LIN {X 121.388,Y 125.417,Z 54.000,A 180.000,B 0.000,C 180.000} C_DIS
LIN {X 121.209,Y 125.491,Z 54.000,A 180.000,B 0.000,C 180.000} C_DIS
LIN {X 120.852,Y 125.619,Z 54.000,A 180.000,B 0.000,C 180.000} C_DIS
LIN {X 120.673,Y 125.674,Z 54.000,A 180.000,B 0.000,C 180.000} C_DIS
LIN {X 120.494,Y 125.726,Z 54.000,A 180.000,B 0.000,C 180.000} C_DIS
LIN {X 120.315,Y 125.774,Z 54.000,A 180.000,B 0.000,C 180.000} C_DIS
LIN {X 119.944,Y 125.857,Z 54.000,A 180.000,B 0.000,C 180.000} C_DIS
LIN {X 119.779,Y 125.886,Z 54.000,A 180.000,B 0.000,C 180.000} C_DIS
LIN {X 119.600,Y 125.914,Z 54.000,A 180.000,B 0.000,C 180.000} C_DIS
LIN {X 119.422,Y 125.941,Z 54.000,A 180.000,B 0.000,C 180.000} C_DIS
LIN {X 119.064,Y 125.975,Z 54.000,A 180.000,B 0.000,C 180.000} C_DIS
LIN {X 118.885,Y 125.987,Z 54.000,A 180.000,B 0.000,C 180.000} C_DIS
LIN {X 118.528,Y 125.998,Z 54.000,A 180.000,B 0.000,C 180.000} C_DIS
LIN {X 118.349,Y 125.994,Z 54.000,A 180.000,B 0.000,C 180.000} C_DIS
LIN {X 118.170,Y 125.988,Z 54.000,A 180.000,B 0.000,C 180.000} C_DIS
LIN {X 117.991,Y 125.980,Z 54.000,A 180.000,B 0.000,C 180.000} C_DIS
LIN {X 117.634,Y 125.947,Z 54.000,A 180.000,B 0.000,C 180.000} C_DIS
LIN {X 117.455,Y 125.923,Z 54.000,A 180.000,B 0.000,C 180.000} C_DIS
LIN {X 117.098,Y 125.866,Z 54.000,A 180.000,B 0.000,C 180.000} C_DIS
LIN {X 117.056,Y 125.857,Z 54.000,A 180.000,B 0.000,C 180.000} C_DIS
LIN {X 116.740,Y 125.787,Z 54.000,A 180.000,B 0.000,C 180.000} C_DIS
LIN {X 116.561,Y 125.742,Z 54.000,A 180.000,B 0.000,C 180.000} C_DIS
LIN {X 116.267,Y 125.656,Z 54.000,A 180.000,B 0.000,C 180.000} C_DIS
LIN {X 116.204,Y 125.638,Z 54.000,A 180.000,B 0.000,C 180.000} C_DIS
LIN {X 116.025,Y 125.575,Z 54.000,A 180.000,B 0.000,C 180.000} C_DIS
LIN {X 115.816,Y 125.500,Z 54.000,A 180.000,B 0.000,C 180.000} C_DIS
LIN {X 115.667,Y 125.441,Z 54.000,A 180.000,B 0.000,C 180.000} C_DIS
LIN {X 115.310,Y 125.286,Z 54.000,A 180.000,B 0.000,C 180.000} C_DIS
LIN {X 115.131,Y 125.195,Z 54.000,A 180.000,B 0.000,C 180.000} C_DIS
LIN {X 114.952,Y 125.104,Z 54.000,A 180.000,B 0.000,C 180.000} C_DIS
LIN {X 114.774,Y 125.004,Z 54.000,A 180.000,B 0.000,C 180.000} C_DIS
LIN {X 114.595,Y 124.898,Z 54.000,A 180.000,B 0.000,C 180.000} C_DIS
LIN {X 114.416,Y 124.787,Z 54.000,A 180.000,B 0.000,C 180.000} C_DIS
LIN {X 114.150,Y 124.606,Z 54.000,A 180.000,B 0.000,C 180.000} C_DIS
LIN {X 114.058,Y 124.540,Z 54.000,A 180.000,B 0.000,C 180.000} C_DIS
LIN {X 113.880,Y 124.402,Z 54.000,A 180.000,B 0.000,C 180.000} C_DIS
LIN {X 113.701,Y 124.261,Z 54.000,A 180.000,B 0.000,C 180.000} C_DIS
LIN {X 113.484,Y 124.070,Z 54.000,A 180.000,B 0.000,C 180.000} C_DIS
LIN {X 113.343,Y 123.943,Z 54.000,A 180.000,B 0.000,C 180.000} C_DIS
LIN {X 113.112,Y 123.712,Z 54.000,A 180.000,B 0.000,C 180.000} C_DIS
LIN {X 112.986,Y 123.579,Z 54.000,A 180.000,B 0.000,C 180.000} C_DIS
LIN {X 112.788,Y 123.354,Z 54.000,A 180.000,B 0.000,C 180.000} C_DIS
LIN {X 112.641,Y 123.176,Z 54.000,A 180.000,B 0.000,C 180.000} C_DIS
LIN {X 112.450,Y 122.928,Z 54.000,A 180.000,B 0.000,C 180.000} C_DIS
LIN {X 112.373,Y 122.818,Z 54.000,A 180.000,B 0.000,C 180.000} C_DIS
LIN {X 112.251,Y 122.639,Z 54.000,A 180.000,B 0.000,C 180.000} C_DIS
LIN {X 112.135,Y 122.461,Z 54.000,A 180.000,B 0.000,C 180.000} C_DIS
LIN {X 112.029,Y 122.282,Z 54.000,A 180.000,B 0.000,C 180.000} C_DIS
LIN {X 111.924,Y 122.103,Z 54.000,A 180.000,B 0.000,C 180.000} C_DIS
LIN {X 111.734,Y 121.731,Z 54.000,A 180.000,B 0.000,C 180.000} C_DIS
LIN {X 111.660,Y 121.567,Z 54.000,A 180.000,B 0.000,C 180.000} C_DIS
LIN {X 111.556,Y 121.325,Z 54.000,A 180.000,B 0.000,C 180.000} C_DIS
LIN {X 111.509,Y 121.209,Z 54.000,A 180.000,B 0.000,C 180.000} C_DIS
LIN {X 111.377,Y 120.841,Z 54.000,A 180.000,B 0.000,C 180.000} C_DIS
LIN {X 111.326,Y 120.673,Z 54.000,A 180.000,B 0.000,C 180.000} C_DIS
LIN {X 111.274,Y 120.494,Z 54.000,A 180.000,B 0.000,C 180.000} C_DIS
LIN {X 111.226,Y 120.315,Z 54.000,A 180.000,B 0.000,C 180.000} C_DIS
LIN {X 111.146,Y 119.958,Z 54.000,A 180.000,B 0.000,C 180.000} C_DIS
LIN {X 111.114,Y 119.779,Z 54.000,A 180.000,B 0.000,C 180.000} C_DIS
LIN {X 111.086,Y 119.600,Z 54.000,A 180.000,B 0.000,C 180.000} C_DIS
LIN {X 111.059,Y 119.422,Z 54.000,A 180.000,B 0.000,C 180.000} C_DIS
LIN {X 111.019,Y 119.006,Z 54.000,A 180.000,B 0.000,C 180.000} C_DIS
LIN {X 111.013,Y 118.885,Z 54.000,A 180.000,B 0.000,C 180.000} C_DIS
LIN {X 111.002,Y 118.528,Z 54.000,A 180.000,B 0.000,C 180.000} C_DIS
LIN {X 111.006,Y 118.349,Z 54.000,A 180.000,B 0.000,C 180.000} C_DIS
LIN {X 111.012,Y 118.170,Z 54.000,A 180.000,B 0.000,C 180.000} C_DIS
LIN {X 111.019,Y 117.994,Z 54.000,A 180.000,B 0.000,C 180.000} C_DIS
LIN {X 111.053,Y 117.634,Z 54.000,A 180.000,B 0.000,C 180.000} C_DIS
LIN {X 111.077,Y 117.455,Z 54.000,A 180.000,B 0.000,C 180.000} C_DIS
LIN {X 111.134,Y 117.098,Z 54.000,A 180.000,B 0.000,C 180.000} C_DIS
LIN {X 111.173,Y 116.919,Z 54.000,A 180.000,B 0.000,C 180.000} C_DIS
LIN {X 111.213,Y 116.740,Z 54.000,A 180.000,B 0.000,C 180.000} C_DIS
LIN {X 111.258,Y 116.561,Z 54.000,A 180.000,B 0.000,C 180.000} C_DIS
LIN {X 111.362,Y 116.204,Z 54.000,A 180.000,B 0.000,C 180.000} C_DIS
LIN {X 111.377,Y 116.159,Z 54.000,A 180.000,B 0.000,C 180.000} C_DIS
LIN {X 111.489,Y 115.846,Z 54.000,A 180.000,B 0.000,C 180.000} C_DIS
LIN {X 111.556,Y 115.675,Z 54.000,A 180.000,B 0.000,C 180.000} C_DIS
LIN {X 111.714,Y 115.310,Z 54.000,A 180.000,B 0.000,C 180.000} C_DIS
LIN {X 111.734,Y 115.269,Z 54.000,A 180.000,B 0.000,C 180.000} C_DIS
LIN {X 111.913,Y 114.918,Z 54.000,A 180.000,B 0.000,C 180.000} C_DIS
LIN {X 111.996,Y 114.774,Z 54.000,A 180.000,B 0.000,C 180.000} C_DIS
LIN {X 112.102,Y 114.595,Z 54.000,A 180.000,B 0.000,C 180.000} C_DIS
LIN {X 112.213,Y 114.416,Z 54.000,A 180.000,B 0.000,C 180.000} C_DIS
LIN {X 112.335,Y 114.237,Z 54.000,A 180.000,B 0.000,C 180.000} C_DIS
LIN {X 112.450,Y 114.072,Z 54.000,A 180.000,B 0.000,C 180.000} C_DIS
LIN {X 112.628,Y 113.841,Z 54.000,A 180.000,B 0.000,C 180.000} C_DIS
LIN {X 112.739,Y 113.701,Z 54.000,A 180.000,B 0.000,C 180.000} C_DIS
LIN {X 112.986,Y 113.421,Z 54.000,A 180.000,B 0.000,C 180.000} C_DIS
LIN {X 113.057,Y 113.343,Z 54.000,A 180.000,B 0.000,C 180.000} C_DIS
LIN {X 113.343,Y 113.057,Z 54.000,A 180.000,B 0.000,C 180.000} C_DIS
LIN {X 113.421,Y 112.986,Z 54.000,A 180.000,B 0.000,C 180.000} C_DIS
LIN {X 113.701,Y 112.739,Z 54.000,A 180.000,B 0.000,C 180.000} C_DIS
LIN {X 113.841,Y 112.628,Z 54.000,A 180.000,B 0.000,C 180.000} C_DIS
LIN {X 114.072,Y 112.450,Z 54.000,A 180.000,B 0.000,C 180.000} C_DIS
LIN {X 114.237,Y 112.335,Z 54.000,A 180.000,B 0.000,C 180.000} C_DIS
LIN {X 114.416,Y 112.213,Z 54.000,A 180.000,B 0.000,C 180.000} C_DIS
LIN {X 114.595,Y 112.102,Z 54.000,A 180.000,B 0.000,C 180.000} C_DIS
LIN {X 114.774,Y 111.996,Z 54.000,A 180.000,B 0.000,C 180.000} C_DIS
LIN {X 114.918,Y 111.913,Z 54.000,A 180.000,B 0.000,C 180.000} C_DIS
LIN {X 115.269,Y 111.734,Z 54.000,A 180.000,B 0.000,C 180.000} C_DIS
LIN {X 115.310,Y 111.714,Z 54.000,A 180.000,B 0.000,C 180.000} C_DIS
LIN {X 115.675,Y 111.556,Z 54.000,A 180.000,B 0.000,C 180.000} C_DIS
LIN {X 115.846,Y 111.489,Z 54.000,A 180.000,B 0.000,C 180.000} C_DIS
LIN {X 116.159,Y 111.377,Z 54.000,A 180.000,B 0.000,C 180.000} C_DIS
LIN {X 116.204,Y 111.362,Z 54.000,A 180.000,B 0.000,C 180.000} C_DIS
LIN {X 116.561,Y 111.258,Z 54.000,A 180.000,B 0.000,C 180.000} C_DIS
LIN {X 116.740,Y 111.213,Z 54.000,A 180.000,B 0.000,C 180.000} C_DIS
LIN {X 116.919,Y 111.173,Z 54.000,A 180.000,B 0.000,C 180.000} C_DIS
LIN {X 117.098,Y 111.134,Z 54.000,A 180.000,B 0.000,C 180.000} C_DIS
LIN {X 117.455,Y 111.077,Z 54.000,A 180.000,B 0.000,C 180.000} C_DIS
LIN {X 117.634,Y 111.053,Z 54.000,A 180.000,B 0.000,C 180.000} C_DIS
LIN {X 117.994,Y 111.019,Z 54.000,A 180.000,B 0.000,C 180.000} C_DIS
LIN {X 118.170,Y 111.012,Z 54.000,A 180.000,B 0.000,C 180.000} C_DIS
LIN {X 118.349,Y 111.006,Z 54.000,A 180.000,B 0.000,C 180.000} C_DIS
LIN {X 118.528,Y 111.002,Z 54.000,A 180.000,B 0.000,C 180.000} C_DIS
LIN {X 118.885,Y 111.013,Z 54.000,A 180.000,B 0.000,C 180.000} C_DIS
LIN {X 119.006,Y 111.019,Z 54.000,A 180.000,B 0.000,C 180.000} C_DIS
LIN {X 119.422,Y 111.059,Z 54.000,A 180.000,B 0.000,C 180.000} C_DIS
LIN {X 119.600,Y 111.086,Z 54.000,A 180.000,B 0.000,C 180.000} C_DIS
LIN {X 119.779,Y 111.114,Z 54.000,A 180.000,B 0.000,C 180.000} C_DIS
LIN {X 119.958,Y 111.146,Z 54.000,A 180.000,B 0.000,C 180.000} C_DIS
LIN {X 120.315,Y 111.226,Z 54.000,A 180.000,B 0.000,C 180.000} C_DIS
LIN {X 120.494,Y 111.274,Z 54.000,A 180.000,B 0.000,C 180.000} C_DIS
LIN {X 120.673,Y 111.326,Z 54.000,A 180.000,B 0.000,C 180.000} C_DIS
LIN {X 120.841,Y 111.377,Z 54.000,A 180.000,B 0.000,C 180.000} C_DIS
LIN {X 121.209,Y 111.509,Z 54.000,A 180.000,B 0.000,C 180.000} C_DIS
LIN {X 121.325,Y 111.556,Z 54.000,A 180.000,B 0.000,C 180.000} C_DIS
LIN {X 121.567,Y 111.660,Z 54.000,A 180.000,B 0.000,C 180.000} C_DIS
LIN {X 121.731,Y 111.734,Z 54.000,A 180.000,B 0.000,C 180.000} C_DIS
LIN {X 122.103,Y 111.924,Z 54.000,A 180.000,B 0.000,C 180.000} C_DIS
LIN {X 122.282,Y 112.029,Z 54.000,A 180.000,B 0.000,C 180.000} C_DIS
LIN {X 122.461,Y 112.135,Z 54.000,A 180.000,B 0.000,C 180.000} C_DIS
LIN {X 122.639,Y 112.251,Z 54.000,A 180.000,B 0.000,C 180.000} C_DIS
LIN {X 122.818,Y 112.373,Z 54.000,A 180.000,B 0.000,C 180.000} C_DIS
LIN {X 122.928,Y 112.450,Z 54.000,A 180.000,B 0.000,C 180.000} C_DIS
LIN {X 123.176,Y 112.641,Z 54.000,A 180.000,B 0.000,C 180.000} C_DIS
LIN {X 123.354,Y 112.788,Z 54.000,A 180.000,B 0.000,C 180.000} C_DIS
LIN {X 123.579,Y 112.986,Z 54.000,A 180.000,B 0.000,C 180.000} C_DIS
LIN {X 123.712,Y 113.112,Z 54.000,A 180.000,B 0.000,C 180.000} C_DIS
LIN {X 123.943,Y 113.343,Z 54.000,A 180.000,B 0.000,C 180.000} C_DIS
LIN {X 124.070,Y 113.484,Z 54.000,A 180.000,B 0.000,C 180.000} C_DIS
LIN {X 124.261,Y 113.701,Z 54.000,A 180.000,B 0.000,C 180.000} C_DIS
LIN {X 124.402,Y 113.880,Z 54.000,A 180.000,B 0.000,C 180.000} C_DIS
LIN {X 124.540,Y 114.058,Z 54.000,A 180.000,B 0.000,C 180.000} C_DIS
LIN {X 124.606,Y 114.150,Z 54.000,A 180.000,B 0.000,C 180.000} C_DIS
LIN {X 124.787,Y 114.416,Z 54.000,A 180.000,B 0.000,C 180.000} C_DIS
LIN {X 124.898,Y 114.595,Z 54.000,A 180.000,B 0.000,C 180.000} C_DIS
LIN {X 125.004,Y 114.774,Z 54.000,A 180.000,B 0.000,C 180.000} C_DIS
LIN {X 125.104,Y 114.952,Z 54.000,A 180.000,B 0.000,C 180.000} C_DIS
LIN {X 125.195,Y 115.131,Z 54.000,A 180.000,B 0.000,C 180.000} C_DIS
LIN {X 125.286,Y 115.310,Z 54.000,A 180.000,B 0.000,C 180.000} C_DIS
LIN {X 125.441,Y 115.667,Z 54.000,A 180.000,B 0.000,C 180.000} C_DIS
LIN {X 125.500,Y 115.816,Z 54.000,A 180.000,B 0.000,C 180.000} C_DIS
LIN {X 125.575,Y 116.025,Z 54.000,A 180.000,B 0.000,C 180.000} C_DIS
LIN {X 125.638,Y 116.204,Z 54.000,A 180.000,B 0.000,C 180.000} C_DIS
LIN {X 125.742,Y 116.561,Z 54.000,A 180.000,B 0.000,C 180.000} C_DIS
LIN {X 125.787,Y 116.740,Z 54.000,A 180.000,B 0.000,C 180.000} C_DIS
LIN {X 125.857,Y 117.056,Z 54.000,A 180.000,B 0.000,C 180.000} C_DIS
LIN {X 125.866,Y 117.098,Z 54.000,A 180.000,B 0.000,C 180.000} C_DIS
LIN {X 125.923,Y 117.455,Z 54.000,A 180.000,B 0.000,C 180.000} C_DIS
LIN {X 125.947,Y 117.634,Z 54.000,A 180.000,B 0.000,C 180.000} C_DIS
LIN {X 125.980,Y 117.991,Z 54.000,A 180.000,B 0.000,C 180.000} C_DIS
LIN {X 125.988,Y 118.170,Z 54.000,A 180.000,B 0.000,C 180.000} C_DIS
LIN {X 125.994,Y 118.349,Z 54.000,A 180.000,B 0.000,C 180.000} C_DIS
LIN {X 125.998,Y 118.528,Z 54.000,A 180.000,B 0.000,C 180.000} C_DIS
LIN {X 125.987,Y 118.885,Z 54.000,A 180.000,B 0.000,C 180.000} C_DIS
LIN {X 125.975,Y 119.064,Z 54.000,A 180.000,B 0.000,C 180.000} C_DIS
LIN {X 125.941,Y 119.422,Z 54.000,A 180.000,B 0.000,C 180.000} C_DIS
LIN {X 125.914,Y 119.600,Z 54.000,A 180.000,B 0.000,C 180.000} C_DIS
LIN {X 125.886,Y 119.779,Z 54.000,A 180.000,B 0.000,C 180.000} C_DIS
LIN {X 125.857,Y 119.944,Z 54.000,A 180.000,B 0.000,C 180.000} C_DIS
LIN {X 125.774,Y 120.315,Z 54.000,A 180.000,B 0.000,C 180.000} C_DIS
LIN {X 125.726,Y 120.494,Z 54.000,A 180.000,B 0.000,C 180.000} C_DIS
LIN {X 125.674,Y 120.673,Z 54.000,A 180.000,B 0.000,C 180.000} C_DIS
LIN {X 125.619,Y 120.852,Z 54.000,A 180.000,B 0.000,C 180.000} C_DIS
LIN {X 125.491,Y 121.209,Z 54.000,A 180.000,B 0.000,C 180.000} C_DIS
LIN {X 125.417,Y 121.388,Z 54.000,A 180.000,B 0.000,C 180.000} C_DIS
LIN {X 125.321,Y 121.610,Z 54.000,A 180.000,B 0.000,C 180.000} C_DIS
LIN {X 125.258,Y 121.746,Z 54.000,A 180.000,B 0.000,C 180.000} C_DIS
LIN {X 125.076,Y 122.103,Z 54.000,A 180.000,B 0.000,C 180.000} C_DIS
LIN {X 124.971,Y 122.282,Z 54.000,A 180.000,B 0.000,C 180.000} C_DIS
LIN {X 124.939,Y 122.336,Z 54.000,A 180.000,B 0.000,C 180.000} C_DIS
; Link Move Starts
LIN {X 124.773,Y 122.604,Z 54.000,A 180.000,B 0.000,C 180.000} C_DIS
LIN {X 124.596,Y 122.864,Z 53.999,A 180.000,B 0.000,C 180.000} C_DIS
LIN {X 124.406,Y 123.115,Z 53.998,A 180.000,B 0.000,C 180.000} C_DIS
LIN {X 124.207,Y 123.360,Z 53.996,A 180.000,B 0.000,C 180.000} C_DIS
LIN {X 123.999,Y 123.596,Z 53.994,A 180.000,B 0.000,C 180.000} C_DIS
LIN {X 123.778,Y 123.821,Z 53.991,A 180.000,B 0.000,C 180.000} C_DIS
LIN {X 123.551,Y 124.039,Z 53.988,A 180.000,B 0.000,C 180.000} C_DIS
LIN {X 123.315,Y 124.247,Z 53.985,A 180.000,B 0.000,C 180.000} C_DIS
LIN {X 123.068,Y 124.443,Z 53.981,A 180.000,B 0.000,C 180.000} C_DIS
LIN {X 122.814,Y 124.630,Z 53.977,A 180.000,B 0.000,C 180.000} C_DIS
LIN {X 122.554,Y 124.807,Z 53.972,A 180.000,B 0.000,C 180.000} C_DIS
LIN {X 122.420,Y 124.890,Z 53.969,A 180.000,B 0.000,C 180.000} C_DIS
LIN {X 122.284,Y 124.970,Z 53.967,A 180.000,B 0.000,C 180.000} C_DIS
LIN {X 122.149,Y 125.050,Z 53.964,A 180.000,B 0.000,C 180.000} C_DIS
LIN {X 122.009,Y 125.124,Z 53.961,A 180.000,B 0.000,C 180.000} C_DIS
LIN {X 121.869,Y 125.195,Z 53.959,A 180.000,B 0.000,C 180.000} C_DIS
LIN {X 121.729,Y 125.267,Z 53.956,A 180.000,B 0.000,C 180.000} C_DIS
LIN {X 121.585,Y 125.332,Z 53.952,A 180.000,B 0.000,C 180.000} C_DIS
LIN {X 121.441,Y 125.394,Z 53.949,A 180.000,B 0.000,C 180.000} C_DIS
LIN {X 121.296,Y 125.457,Z 53.946,A 180.000,B 0.000,C 180.000} C_DIS
LIN {X 121.149,Y 125.512,Z 53.943,A 180.000,B 0.000,C 180.000} C_DIS
LIN {X 121.001,Y 125.566,Z 53.939,A 180.000,B 0.000,C 180.000} C_DIS
LIN {X 120.852,Y 125.619,Z 53.936,A 180.000,B 0.000,C 180.000} C_DIS
LIN {X 120.702,Y 125.665,Z 53.932,A 180.000,B 0.000,C 180.000} C_DIS
LIN {X 120.551,Y 125.709,Z 53.928,A 180.000,B 0.000,C 180.000} C_DIS
LIN {X 120.399,Y 125.753,Z 53.925,A 180.000,B 0.000,C 180.000} C_DIS
LIN {X 120.246,Y 125.790,Z 53.921,A 180.000,B 0.000,C 180.000} C_DIS
LIN {X 120.092,Y 125.824,Z 53.917,A 180.000,B 0.000,C 180.000} C_DIS
LIN {X 119.939,Y 125.858,Z 53.913,A 180.000,B 0.000,C 180.000} C_DIS
LIN {X 119.784,Y 125.885,Z 53.909,A 180.000,B 0.000,C 180.000} C_DIS
LIN {X 119.628,Y 125.910,Z 53.905,A 180.000,B 0.000,C 180.000} C_DIS
LIN {X 119.472,Y 125.934,Z 53.900,A 180.000,B 0.000,C 180.000} C_DIS
LIN {X 119.316,Y 125.951,Z 53.896,A 180.000,B 0.000,C 180.000} C_DIS
LIN {X 119.159,Y 125.966,Z 53.892,A 180.000,B 0.000,C 180.000} C_DIS
LIN {X 119.002,Y 125.981,Z 53.887,A 180.000,B 0.000,C 180.000} C_DIS
LIN {X 118.845,Y 125.988,Z 53.883,A 180.000,B 0.000,C 180.000} C_DIS
LIN {X 118.687,Y 125.993,Z 53.878,A 180.000,B 0.000,C 180.000} C_DIS
LIN {X 118.530,Y 125.998,Z 53.873,A 180.000,B 0.000,C 180.000} C_DIS
LIN {X 118.373,Y 125.995,Z 53.869,A 180.000,B 0.000,C 180.000} C_DIS
LIN {X 118.215,Y 125.990,Z 53.864,A 180.000,B 0.000,C 180.000} C_DIS
LIN {X 118.058,Y 125.985,Z 53.859,A 180.000,B 0.000,C 180.000} C_DIS
LIN {X 117.901,Y 125.972,Z 53.854,A 180.000,B 0.000,C 180.000} C_DIS
LIN {X 117.822,Y 125.964,Z 53.851,A 180.000,B 0.000,C 180.000} C_DIS
LIN {X 117.744,Y 125.957,Z 53.849,A 180.000,B 0.000,C 180.000} C_DIS
LIN {X 117.666,Y 125.950,Z 53.846,A 180.000,B 0.000,C 180.000} C_DIS
LIN {X 117.587,Y 125.942,Z 53.844,A 180.000,B 0.000,C 180.000} C_DIS
LIN {X 117.509,Y 125.932,Z 53.841,A 180.000,B 0.000,C 180.000} C_DIS
LIN {X 117.431,Y 125.919,Z 53.839,A 180.000,B 0.000,C 180.000} C_DIS
LIN {X 117.354,Y 125.907,Z 53.836,A 180.000,B 0.000,C 180.000} C_DIS
LIN {X 117.198,Y 125.882,Z 53.831,A 180.000,B 0.000,C 180.000} C_DIS
LIN {X 117.120,Y 125.870,Z 53.828,A 180.000,B 0.000,C 180.000} C_DIS
LIN {X 117.043,Y 125.854,Z 53.825,A 180.000,B 0.000,C 180.000} C_DIS
LIN {X 116.889,Y 125.820,Z 53.820,A 180.000,B 0.000,C 180.000} C_DIS
LIN {X 116.736,Y 125.786,Z 53.815,A 180.000,B 0.000,C 180.000} C_DIS
LIN {X 116.659,Y 125.768,Z 53.812,A 180.000,B 0.000,C 180.000} C_DIS
LIN {X 116.583,Y 125.748,Z 53.809,A 180.000,B 0.000,C 180.000} C_DIS
LIN {X 116.507,Y 125.726,Z 53.806,A 180.000,B 0.000,C 180.000} C_DIS
LIN {X 116.356,Y 125.682,Z 53.801,A 180.000,B 0.000,C 180.000} C_DIS
LIN {X 116.205,Y 125.638,Z 53.796,A 180.000,B 0.000,C 180.000} C_DIS
LIN {X 116.130,Y 125.613,Z 53.793,A 180.000,B 0.000,C 180.000} C_DIS
LIN {X 115.982,Y 125.559,Z 53.787,A 180.000,B 0.000,C 180.000} C_DIS
LIN {X 115.908,Y 125.533,Z 53.785,A 180.000,B 0.000,C 180.000} C_DIS
LIN {X 115.759,Y 125.479,Z 53.779,A 180.000,B 0.000,C 180.000} C_DIS
LIN {X 115.687,Y 125.449,Z 53.776,A 180.000,B 0.000,C 180.000} C_DIS
LIN {X 115.614,Y 125.418,Z 53.774,A 180.000,B 0.000,C 180.000} C_DIS
LIN {X 115.470,Y 125.355,Z 53.768,A 180.000,B 0.000,C 180.000} C_DIS
LIN {X 115.325,Y 125.293,Z 53.763,A 180.000,B 0.000,C 180.000} C_DIS
LIN {X 115.255,Y 125.258,Z 53.760,A 180.000,B 0.000,C 180.000} C_DIS
LIN {X 115.114,Y 125.187,Z 53.754,A 180.000,B 0.000,C 180.000} C_DIS
LIN {X 115.044,Y 125.151,Z 53.752,A 180.000,B 0.000,C 180.000} C_DIS
LIN {X 114.904,Y 125.080,Z 53.746,A 180.000,B 0.000,C 180.000} C_DIS
LIN {X 114.835,Y 125.040,Z 53.743,A 180.000,B 0.000,C 180.000} C_DIS
LIN {X 114.768,Y 125.000,Z 53.741,A 180.000,B 0.000,C 180.000} C_DIS
LIN {X 114.632,Y 124.920,Z 53.735,A 180.000,B 0.000,C 180.000} C_DIS
LIN {X 114.496,Y 124.840,Z 53.730,A 180.000,B 0.000,C 180.000} C_DIS
LIN {X 114.431,Y 124.797,Z 53.727,A 180.000,B 0.000,C 180.000} C_DIS
LIN {X 114.300,Y 124.708,Z 53.721,A 180.000,B 0.000,C 180.000} C_DIS
LIN {X 114.235,Y 124.664,Z 53.719,A 180.000,B 0.000,C 180.000} C_DIS
LIN {X 114.105,Y 124.575,Z 53.713,A 180.000,B 0.000,C 180.000} C_DIS
LIN {X 114.042,Y 124.528,Z 53.710,A 180.000,B 0.000,C 180.000} C_DIS
LIN {X 113.980,Y 124.479,Z 53.708,A 180.000,B 0.000,C 180.000} C_DIS
LIN {X 113.855,Y 124.383,Z 53.702,A 180.000,B 0.000,C 180.000} C_DIS
LIN {X 113.731,Y 124.286,Z 53.697,A 180.000,B 0.000,C 180.000} C_DIS
LIN {X 113.671,Y 124.235,Z 53.694,A 180.000,B 0.000,C 180.000} C_DIS
LIN {X 113.553,Y 124.131,Z 53.688,A 180.000,B 0.000,C 180.000} C_DIS
LIN {X 113.494,Y 124.079,Z 53.686,A 180.000,B 0.000,C 180.000} C_DIS
LIN {X 113.376,Y 123.975,Z 53.680,A 180.000,B 0.000,C 180.000} C_DIS
LIN {X 113.320,Y 123.919,Z 53.677,A 180.000,B 0.000,C 180.000} C_DIS
LIN {X 113.208,Y 123.808,Z 53.672,A 180.000,B 0.000,C 180.000} C_DIS
LIN {X 113.097,Y 123.697,Z 53.666,A 180.000,B 0.000,C 180.000} C_DIS
LIN {X 113.041,Y 123.641,Z 53.664,A 180.000,B 0.000,C 180.000} C_DIS
LIN {X 112.989,Y 123.582,Z 53.661,A 180.000,B 0.000,C 180.000} C_DIS
LIN {X 112.728,Y 123.287,Z 53.647,A 180.000,B 0.000,C 180.000} C_DIS
LIN {X 112.680,Y 123.225,Z 53.644,A 180.000,B 0.000,C 180.000} C_DIS
LIN {X 112.583,Y 123.101,Z 53.639,A 180.000,B 0.000,C 180.000} C_DIS
LIN {X 112.438,Y 122.914,Z 53.631,A 180.000,B 0.000,C 180.000} C_DIS
LIN {X 112.394,Y 122.849,Z 53.628,A 180.000,B 0.000,C 180.000} C_DIS
LIN {X 112.172,Y 122.523,Z 53.614,A 180.000,B 0.000,C 180.000} C_DIS
LIN {X 112.132,Y 122.456,Z 53.611,A 180.000,B 0.000,C 180.000} C_DIS
LIN {X 112.011,Y 122.252,Z 53.603,A 180.000,B 0.000,C 180.000} C_DIS
LIN {X 111.931,Y 122.117,Z 53.598,A 180.000,B 0.000,C 180.000} C_DIS
LIN {X 111.895,Y 122.047,Z 53.595,A 180.000,B 0.000,C 180.000} C_DIS
LIN {X 111.716,Y 121.696,Z 53.581,A 180.000,B 0.000,C 180.000} C_DIS
LIN {X 111.685,Y 121.624,Z 53.578,A 180.000,B 0.000,C 180.000} C_DIS
LIN {X 111.529,Y 121.262,Z 53.565,A 180.000,B 0.000,C 180.000} C_DIS
LIN {X 111.502,Y 121.188,Z 53.562,A 180.000,B 0.000,C 180.000} C_DIS
LIN {X 111.368,Y 120.818,Z 53.548,A 180.000,B 0.000,C 180.000} C_DIS
LIN {X 111.346,Y 120.742,Z 53.545,A 180.000,B 0.000,C 180.000} C_DIS
LIN {X 111.259,Y 120.440,Z 53.534,A 180.000,B 0.000,C 180.000} C_DIS
LIN {X 111.237,Y 120.364,Z 53.532,A 180.000,B 0.000,C 180.000} C_DIS
LIN {X 111.151,Y 119.980,Z 53.518,A 180.000,B 0.000,C 180.000} C_DIS
LIN {X 111.134,Y 119.903,Z 53.515,A 180.000,B 0.000,C 180.000} C_DIS
LIN {X 111.072,Y 119.514,Z 53.501,A 180.000,B 0.000,C 180.000} C_DIS
LIN {X 111.060,Y 119.436,Z 53.499,A 180.000,B 0.000,C 180.000} C_DIS
LIN {X 111.023,Y 119.044,Z 53.485,A 180.000,B 0.000,C 180.000} C_DIS
LIN {X 111.016,Y 118.965,Z 53.482,A 180.000,B 0.000,C 180.000} C_DIS
LIN {X 111.003,Y 118.572,Z 53.468,A 180.000,B 0.000,C 180.000} C_DIS
LIN {X 111.001,Y 118.493,Z 53.466,A 180.000,B 0.000,C 180.000} C_DIS
LIN {X 111.014,Y 118.100,Z 53.452,A 180.000,B 0.000,C 180.000} C_DIS
LIN {X 111.017,Y 118.021,Z 53.449,A 180.000,B 0.000,C 180.000} C_DIS
LIN {X 111.054,Y 117.629,Z 53.435,A 180.000,B 0.000,C 180.000} C_DIS
LIN {X 111.062,Y 117.550,Z 53.433,A 180.000,B 0.000,C 180.000} C_DIS
LIN {X 111.123,Y 117.162,Z 53.419,A 180.000,B 0.000,C 180.000} C_DIS
LIN {X 111.137,Y 117.084,Z 53.416,A 180.000,B 0.000,C 180.000} C_DIS
LIN {X 111.222,Y 116.700,Z 53.402,A 180.000,B 0.000,C 180.000} C_DIS
LIN {X 111.240,Y 116.623,Z 53.400,A 180.000,B 0.000,C 180.000} C_DIS
LIN {X 111.306,Y 116.396,Z 53.391,A 180.000,B 0.000,C 180.000} C_DIS
LIN {X 111.350,Y 116.245,Z 53.386,A 180.000,B 0.000,C 180.000} C_DIS
LIN {X 111.373,Y 116.169,Z 53.383,A 180.000,B 0.000,C 180.000} C_DIS
LIN {X 111.506,Y 115.799,Z 53.369,A 180.000,B 0.000,C 180.000} C_DIS
LIN {X 111.534,Y 115.725,Z 53.367,A 180.000,B 0.000,C 180.000} C_DIS
LIN {X 111.628,Y 115.508,Z 53.358,A 180.000,B 0.000,C 180.000} C_DIS
LIN {X 111.690,Y 115.364,Z 53.353,A 180.000,B 0.000,C 180.000} C_DIS
LIN {X 111.723,Y 115.292,Z 53.350,A 180.000,B 0.000,C 180.000} C_DIS
LIN {X 111.901,Y 114.941,Z 53.336,A 180.000,B 0.000,C 180.000} C_DIS
LIN {X 111.938,Y 114.871,Z 53.334,A 180.000,B 0.000,C 180.000} C_DIS
LIN {X 112.018,Y 114.736,Z 53.328,A 180.000,B 0.000,C 180.000} C_DIS
LIN {X 112.139,Y 114.533,Z 53.320,A 180.000,B 0.000,C 180.000} C_DIS
LIN {X 112.180,Y 114.465,Z 53.317,A 180.000,B 0.000,C 180.000} C_DIS
LIN {X 112.401,Y 114.140,Z 53.303,A 180.000,B 0.000,C 180.000} C_DIS
LIN {X 112.447,Y 114.075,Z 53.301,A 180.000,B 0.000,C 180.000} C_DIS
LIN {X 112.543,Y 113.951,Z 53.295,A 180.000,B 0.000,C 180.000} C_DIS
LIN {X 112.688,Y 113.764,Z 53.287,A 180.000,B 0.000,C 180.000} C_DIS
LIN {X 112.737,Y 113.703,Z 53.284,A 180.000,B 0.000,C 180.000} C_DIS
LIN {X 112.894,Y 113.526,Z 53.276,A 180.000,B 0.000,C 180.000} C_DIS
LIN {X 112.998,Y 113.407,Z 53.270,A 180.000,B 0.000,C 180.000} C_DIS
LIN {X 113.051,Y 113.349,Z 53.268,A 180.000,B 0.000,C 180.000} C_DIS
LIN {X 113.162,Y 113.238,Z 53.262,A 180.000,B 0.000,C 180.000} C_DIS
LIN {X 113.329,Y 113.071,Z 53.254,A 180.000,B 0.000,C 180.000} C_DIS
LIN {X 113.386,Y 113.016,Z 53.251,A 180.000,B 0.000,C 180.000} C_DIS
LIN {X 113.563,Y 112.860,Z 53.243,A 180.000,B 0.000,C 180.000} C_DIS
LIN {X 113.682,Y 112.756,Z 53.237,A 180.000,B 0.000,C 180.000} C_DIS
LIN {X 113.742,Y 112.705,Z 53.235,A 180.000,B 0.000,C 180.000} C_DIS
LIN {X 113.866,Y 112.609,Z 53.229,A 180.000,B 0.000,C 180.000} C_DIS
LIN {X 114.053,Y 112.464,Z 53.221,A 180.000,B 0.000,C 180.000} C_DIS
LIN {X 114.116,Y 112.417,Z 53.218,A 180.000,B 0.000,C 180.000} C_DIS
LIN {X 114.312,Y 112.284,Z 53.210,A 180.000,B 0.000,C 180.000} C_DIS
LIN {X 114.442,Y 112.196,Z 53.204,A 180.000,B 0.000,C 180.000} C_DIS
LIN {X 114.508,Y 112.153,Z 53.202,A 180.000,B 0.000,C 180.000} C_DIS
LIN {X 114.644,Y 112.073,Z 53.196,A 180.000,B 0.000,C 180.000} C_DIS
LIN {X 114.779,Y 111.993,Z 53.191,A 180.000,B 0.000,C 180.000} C_DIS
LIN {X 114.847,Y 111.953,Z 53.188,A 180.000,B 0.000,C 180.000} C_DIS
LIN {X 114.916,Y 111.914,Z 53.185,A 180.000,B 0.000,C 180.000} C_DIS
LIN {X 115.056,Y 111.843,Z 53.180,A 180.000,B 0.000,C 180.000} C_DIS
LIN {X 115.196,Y 111.771,Z 53.174,A 180.000,B 0.000,C 180.000} C_DIS
LIN {X 115.267,Y 111.736,Z 53.172,A 180.000,B 0.000,C 180.000} C_DIS
LIN {X 115.338,Y 111.702,Z 53.169,A 180.000,B 0.000,C 180.000} C_DIS
LIN {X 115.482,Y 111.639,Z 53.164,A 180.000,B 0.000,C 180.000} C_DIS
LIN {X 115.555,Y 111.608,Z 53.161,A 180.000,B 0.000,C 180.000} C_DIS
LIN {X 115.627,Y 111.577,Z 53.159,A 180.000,B 0.000,C 180.000} C_DIS
LIN {X 115.699,Y 111.545,Z 53.156,A 180.000,B 0.000,C 180.000} C_DIS
LIN {X 115.772,Y 111.516,Z 53.154,A 180.000,B 0.000,C 180.000} C_DIS
LIN {X 115.846,Y 111.489,Z 53.151,A 180.000,B 0.000,C 180.000} C_DIS
LIN {X 115.920,Y 111.463,Z 53.149,A 180.000,B 0.000,C 180.000} C_DIS
LIN {X 116.069,Y 111.409,Z 53.144,A 180.000,B 0.000,C 180.000} C_DIS
LIN {X 116.217,Y 111.358,Z 53.139,A 180.000,B 0.000,C 180.000} C_DIS
LIN {X 116.369,Y 111.314,Z 53.134,A 180.000,B 0.000,C 180.000} C_DIS
LIN {X 116.520,Y 111.270,Z 53.129,A 180.000,B 0.000,C 180.000} C_DIS
LIN {X 116.672,Y 111.229,Z 53.124,A 180.000,B 0.000,C 180.000} C_DIS
LIN {X 116.826,Y 111.194,Z 53.120,A 180.000,B 0.000,C 180.000} C_DIS
LIN {X 116.979,Y 111.160,Z 53.115,A 180.000,B 0.000,C 180.000} C_DIS
LIN {X 117.133,Y 111.128,Z 53.111,A 180.000,B 0.000,C 180.000} C_DIS
LIN {X 117.289,Y 111.103,Z 53.106,A 180.000,B 0.000,C 180.000} C_DIS
LIN {X 117.445,Y 111.079,Z 53.102,A 180.000,B 0.000,C 180.000} C_DIS
LIN {X 117.601,Y 111.057,Z 53.097,A 180.000,B 0.000,C 180.000} C_DIS
LIN {X 117.757,Y 111.042,Z 53.093,A 180.000,B 0.000,C 180.000} C_DIS
LIN {X 117.914,Y 111.027,Z 53.089,A 180.000,B 0.000,C 180.000} C_DIS
LIN {X 118.071,Y 111.015,Z 53.085,A 180.000,B 0.000,C 180.000} C_DIS
LIN {X 118.229,Y 111.010,Z 53.081,A 180.000,B 0.000,C 180.000} C_DIS
LIN {X 118.386,Y 111.005,Z 53.077,A 180.000,B 0.000,C 180.000} C_DIS
LIN {X 118.544,Y 111.003,Z 53.073,A 180.000,B 0.000,C 180.000} C_DIS
LIN {X 118.701,Y 111.008,Z 53.070,A 180.000,B 0.000,C 180.000} C_DIS
LIN {X 118.858,Y 111.012,Z 53.066,A 180.000,B 0.000,C 180.000} C_DIS
LIN {X 119.016,Y 111.020,Z 53.062,A 180.000,B 0.000,C 180.000} C_DIS
LIN {X 119.172,Y 111.035,Z 53.059,A 180.000,B 0.000,C 180.000} C_DIS
LIN {X 119.329,Y 111.050,Z 53.056,A 180.000,B 0.000,C 180.000} C_DIS
LIN {X 119.486,Y 111.068,Z 53.052,A 180.000,B 0.000,C 180.000} C_DIS
LIN {X 119.641,Y 111.092,Z 53.049,A 180.000,B 0.000,C 180.000} C_DIS
LIN {X 119.797,Y 111.117,Z 53.046,A 180.000,B 0.000,C 180.000} C_DIS
LIN {X 119.952,Y 111.145,Z 53.043,A 180.000,B 0.000,C 180.000} C_DIS
LIN {X 120.106,Y 111.179,Z 53.040,A 180.000,B 0.000,C 180.000} C_DIS
LIN {X 120.259,Y 111.213,Z 53.037,A 180.000,B 0.000,C 180.000} C_DIS
LIN {X 120.412,Y 111.251,Z 53.034,A 180.000,B 0.000,C 180.000} C_DIS
LIN {X 120.564,Y 111.295,Z 53.032,A 180.000,B 0.000,C 180.000} C_DIS
LIN {X 120.715,Y 111.338,Z 53.029,A 180.000,B 0.000,C 180.000} C_DIS
LIN {X 120.865,Y 111.385,Z 53.027,A 180.000,B 0.000,C 180.000} C_DIS
LIN {X 121.161,Y 111.492,Z 53.022,A 180.000,B 0.000,C 180.000} C_DIS
LIN {X 121.453,Y 111.611,Z 53.018,A 180.000,B 0.000,C 180.000} C_DIS
LIN {X 121.741,Y 111.739,Z 53.014,A 180.000,B 0.000,C 180.000} C_DIS
LIN {X 122.021,Y 111.882,Z 53.011,A 180.000,B 0.000,C 180.000} C_DIS
LIN {X 122.296,Y 112.037,Z 53.008,A 180.000,B 0.000,C 180.000} C_DIS
LIN {X 122.565,Y 112.200,Z 53.005,A 180.000,B 0.000,C 180.000} C_DIS
LIN {X 122.826,Y 112.378,Z 53.003,A 180.000,B 0.000,C 180.000} C_DIS
LIN {X 123.078,Y 112.566,Z 53.002,A 180.000,B 0.000,C 180.000} C_DIS
LIN {X 123.325,Y 112.762,Z 53.001,A 180.000,B 0.000,C 180.000} C_DIS
LIN {X 123.561,Y 112.970,Z 53.000,A 180.000,B 0.000,C 180.000} C_DIS
LIN {X 123.729,Y 113.130,Z 53.000,A 180.000,B 0.000,C 180.000} C_DIS
; Cutting Move Starts
LIN {X 123.943,Y 113.343,Z 53.000,A 180.000,B 0.000,C 180.000} C_DIS
LIN {X 124.070,Y 113.484,Z 53.000,A 180.000,B 0.000,C 180.000} C_DIS
LIN {X 124.261,Y 113.701,Z 53.000,A 180.000,B 0.000,C 180.000} C_DIS
LIN {X 124.402,Y 113.880,Z 53.000,A 180.000,B 0.000,C 180.000} C_DIS
LIN {X 124.540,Y 114.058,Z 53.000,A 180.000,B 0.000,C 180.000} C_DIS
LIN {X 124.606,Y 114.150,Z 53.000,A 180.000,B 0.000,C 180.000} C_DIS
LIN {X 124.787,Y 114.416,Z 53.000,A 180.000,B 0.000,C 180.000} C_DIS
LIN {X 124.898,Y 114.595,Z 53.000,A 180.000,B 0.000,C 180.000} C_DIS
LIN {X 125.004,Y 114.774,Z 53.000,A 180.000,B 0.000,C 180.000} C_DIS
LIN {X 125.104,Y 114.952,Z 53.000,A 180.000,B 0.000,C 180.000} C_DIS
LIN {X 125.195,Y 115.131,Z 53.000,A 180.000,B 0.000,C 180.000} C_DIS
LIN {X 125.286,Y 115.310,Z 53.000,A 180.000,B 0.000,C 180.000} C_DIS
LIN {X 125.441,Y 115.667,Z 53.000,A 180.000,B 0.000,C 180.000} C_DIS
LIN {X 125.500,Y 115.816,Z 53.000,A 180.000,B 0.000,C 180.000} C_DIS
LIN {X 125.575,Y 116.025,Z 53.000,A 180.000,B 0.000,C 180.000} C_DIS
LIN {X 125.638,Y 116.204,Z 53.000,A 180.000,B 0.000,C 180.000} C_DIS
LIN {X 125.742,Y 116.561,Z 53.000,A 180.000,B 0.000,C 180.000} C_DIS
LIN {X 125.787,Y 116.740,Z 53.000,A 180.000,B 0.000,C 180.000} C_DIS
LIN {X 125.857,Y 117.056,Z 53.000,A 180.000,B 0.000,C 180.000} C_DIS
LIN {X 125.866,Y 117.098,Z 53.000,A 180.000,B 0.000,C 180.000} C_DIS
LIN {X 125.923,Y 117.455,Z 53.000,A 180.000,B 0.000,C 180.000} C_DIS
LIN {X 125.947,Y 117.634,Z 53.000,A 180.000,B 0.000,C 180.000} C_DIS
LIN {X 125.980,Y 117.991,Z 53.000,A 180.000,B 0.000,C 180.000} C_DIS
LIN {X 125.988,Y 118.170,Z 53.000,A 180.000,B 0.000,C 180.000} C_DIS
LIN {X 125.994,Y 118.349,Z 53.000,A 180.000,B 0.000,C 180.000} C_DIS
LIN {X 125.998,Y 118.528,Z 53.000,A 180.000,B 0.000,C 180.000} C_DIS
LIN {X 125.987,Y 118.885,Z 53.000,A 180.000,B 0.000,C 180.000} C_DIS
LIN {X 125.975,Y 119.064,Z 53.000,A 180.000,B 0.000,C 180.000} C_DIS
LIN {X 125.941,Y 119.422,Z 53.000,A 180.000,B 0.000,C 180.000} C_DIS
LIN {X 125.914,Y 119.600,Z 53.000,A 180.000,B 0.000,C 180.000} C_DIS
LIN {X 125.886,Y 119.779,Z 53.000,A 180.000,B 0.000,C 180.000} C_DIS
LIN {X 125.857,Y 119.944,Z 53.000,A 180.000,B 0.000,C 180.000} C_DIS
LIN {X 125.774,Y 120.315,Z 53.000,A 180.000,B 0.000,C 180.000} C_DIS
LIN {X 125.726,Y 120.494,Z 53.000,A 180.000,B 0.000,C 180.000} C_DIS
LIN {X 125.674,Y 120.673,Z 53.000,A 180.000,B 0.000,C 180.000} C_DIS
LIN {X 125.619,Y 120.852,Z 53.000,A 180.000,B 0.000,C 180.000} C_DIS
LIN {X 125.491,Y 121.209,Z 53.000,A 180.000,B 0.000,C 180.000} C_DIS
LIN {X 125.417,Y 121.388,Z 53.000,A 180.000,B 0.000,C 180.000} C_DIS
LIN {X 125.321,Y 121.610,Z 53.000,A 180.000,B 0.000,C 180.000} C_DIS
LIN {X 125.258,Y 121.746,Z 53.000,A 180.000,B 0.000,C 180.000} C_DIS
LIN {X 125.076,Y 122.103,Z 53.000,A 180.000,B 0.000,C 180.000} C_DIS
LIN {X 124.971,Y 122.282,Z 53.000,A 180.000,B 0.000,C 180.000} C_DIS
LIN {X 124.865,Y 122.461,Z 53.000,A 180.000,B 0.000,C 180.000} C_DIS
LIN {X 124.785,Y 122.587,Z 53.000,A 180.000,B 0.000,C 180.000} C_DIS
LIN {X 124.606,Y 122.850,Z 53.000,A 180.000,B 0.000,C 180.000} C_DIS
LIN {X 124.497,Y 122.997,Z 53.000,A 180.000,B 0.000,C 180.000} C_DIS
LIN {X 124.359,Y 123.176,Z 53.000,A 180.000,B 0.000,C 180.000} C_DIS
LIN {X 124.248,Y 123.313,Z 53.000,A 180.000,B 0.000,C 180.000} C_DIS
LIN {X 124.055,Y 123.533,Z 53.000,A 180.000,B 0.000,C 180.000} C_DIS
LIN {X 123.891,Y 123.709,Z 53.000,A 180.000,B 0.000,C 180.000} C_DIS
LIN {X 123.709,Y 123.891,Z 53.000,A 180.000,B 0.000,C 180.000} C_DIS
LIN {X 123.533,Y 124.055,Z 53.000,A 180.000,B 0.000,C 180.000} C_DIS
LIN {X 123.313,Y 124.248,Z 53.000,A 180.000,B 0.000,C 180.000} C_DIS
LIN {X 123.176,Y 124.359,Z 53.000,A 180.000,B 0.000,C 180.000} C_DIS
LIN {X 122.997,Y 124.497,Z 53.000,A 180.000,B 0.000,C 180.000} C_DIS
LIN {X 122.850,Y 124.606,Z 53.000,A 180.000,B 0.000,C 180.000} C_DIS
LIN {X 122.587,Y 124.785,Z 53.000,A 180.000,B 0.000,C 180.000} C_DIS
LIN {X 122.461,Y 124.865,Z 53.000,A 180.000,B 0.000,C 180.000} C_DIS
LIN {X 122.282,Y 124.971,Z 53.000,A 180.000,B 0.000,C 180.000} C_DIS
LIN {X 122.103,Y 125.076,Z 53.000,A 180.000,B 0.000,C 180.000} C_DIS
LIN {X 121.746,Y 125.258,Z 53.000,A 180.000,B 0.000,C 180.000} C_DIS
LIN {X 121.610,Y 125.321,Z 53.000,A 180.000,B 0.000,C 180.000} C_DIS
LIN {X 121.388,Y 125.417,Z 53.000,A 180.000,B 0.000,C 180.000} C_DIS
LIN {X 121.209,Y 125.491,Z 53.000,A 180.000,B 0.000,C 180.000} C_DIS
LIN {X 120.852,Y 125.619,Z 53.000,A 180.000,B 0.000,C 180.000} C_DIS
LIN {X 120.673,Y 125.674,Z 53.000,A 180.000,B 0.000,C 180.000} C_DIS
LIN {X 120.494,Y 125.726,Z 53.000,A 180.000,B 0.000,C 180.000} C_DIS
LIN {X 120.315,Y 125.774,Z 53.000,A 180.000,B 0.000,C 180.000} C_DIS
LIN {X 119.944,Y 125.857,Z 53.000,A 180.000,B 0.000,C 180.000} C_DIS
LIN {X 119.779,Y 125.886,Z 53.000,A 180.000,B 0.000,C 180.000} C_DIS
LIN {X 119.600,Y 125.914,Z 53.000,A 180.000,B 0.000,C 180.000} C_DIS
LIN {X 119.422,Y 125.941,Z 53.000,A 180.000,B 0.000,C 180.000} C_DIS
LIN {X 119.064,Y 125.975,Z 53.000,A 180.000,B 0.000,C 180.000} C_DIS
LIN {X 118.885,Y 125.987,Z 53.000,A 180.000,B 0.000,C 180.000} C_DIS
LIN {X 118.528,Y 125.998,Z 53.000,A 180.000,B 0.000,C 180.000} C_DIS
LIN {X 118.349,Y 125.994,Z 53.000,A 180.000,B 0.000,C 180.000} C_DIS
LIN {X 118.170,Y 125.988,Z 53.000,A 180.000,B 0.000,C 180.000} C_DIS
LIN {X 117.991,Y 125.980,Z 53.000,A 180.000,B 0.000,C 180.000} C_DIS
LIN {X 117.634,Y 125.947,Z 53.000,A 180.000,B 0.000,C 180.000} C_DIS
LIN {X 117.455,Y 125.923,Z 53.000,A 180.000,B 0.000,C 180.000} C_DIS
LIN {X 117.098,Y 125.866,Z 53.000,A 180.000,B 0.000,C 180.000} C_DIS
LIN {X 117.056,Y 125.857,Z 53.000,A 180.000,B 0.000,C 180.000} C_DIS
LIN {X 116.740,Y 125.787,Z 53.000,A 180.000,B 0.000,C 180.000} C_DIS
LIN {X 116.561,Y 125.742,Z 53.000,A 180.000,B 0.000,C 180.000} C_DIS
LIN {X 116.204,Y 125.638,Z 53.000,A 180.000,B 0.000,C 180.000} C_DIS
LIN {X 116.025,Y 125.575,Z 53.000,A 180.000,B 0.000,C 180.000} C_DIS
LIN {X 115.816,Y 125.500,Z 53.000,A 180.000,B 0.000,C 180.000} C_DIS
LIN {X 115.667,Y 125.441,Z 53.000,A 180.000,B 0.000,C 180.000} C_DIS
LIN {X 115.310,Y 125.286,Z 53.000,A 180.000,B 0.000,C 180.000} C_DIS
LIN {X 115.131,Y 125.195,Z 53.000,A 180.000,B 0.000,C 180.000} C_DIS
LIN {X 114.952,Y 125.104,Z 53.000,A 180.000,B 0.000,C 180.000} C_DIS
LIN {X 114.774,Y 125.004,Z 53.000,A 180.000,B 0.000,C 180.000} C_DIS
LIN {X 114.595,Y 124.898,Z 53.000,A 180.000,B 0.000,C 180.000} C_DIS
LIN {X 114.416,Y 124.787,Z 53.000,A 180.000,B 0.000,C 180.000} C_DIS
LIN {X 114.150,Y 124.606,Z 53.000,A 180.000,B 0.000,C 180.000} C_DIS
LIN {X 114.058,Y 124.540,Z 53.000,A 180.000,B 0.000,C 180.000} C_DIS
LIN {X 113.880,Y 124.402,Z 53.000,A 180.000,B 0.000,C 180.000} C_DIS
LIN {X 113.701,Y 124.261,Z 53.000,A 180.000,B 0.000,C 180.000} C_DIS
LIN {X 113.484,Y 124.070,Z 53.000,A 180.000,B 0.000,C 180.000} C_DIS
LIN {X 113.343,Y 123.943,Z 53.000,A 180.000,B 0.000,C 180.000} C_DIS
LIN {X 113.112,Y 123.712,Z 53.000,A 180.000,B 0.000,C 180.000} C_DIS
LIN {X 112.986,Y 123.579,Z 53.000,A 180.000,B 0.000,C 180.000} C_DIS
LIN {X 112.788,Y 123.354,Z 53.000,A 180.000,B 0.000,C 180.000} C_DIS
LIN {X 112.641,Y 123.176,Z 53.000,A 180.000,B 0.000,C 180.000} C_DIS
LIN {X 112.450,Y 122.928,Z 53.000,A 180.000,B 0.000,C 180.000} C_DIS
LIN {X 112.373,Y 122.818,Z 53.000,A 180.000,B 0.000,C 180.000} C_DIS
LIN {X 112.251,Y 122.639,Z 53.000,A 180.000,B 0.000,C 180.000} C_DIS
LIN {X 112.135,Y 122.461,Z 53.000,A 180.000,B 0.000,C 180.000} C_DIS
LIN {X 112.029,Y 122.282,Z 53.000,A 180.000,B 0.000,C 180.000} C_DIS
LIN {X 111.924,Y 122.103,Z 53.000,A 180.000,B 0.000,C 180.000} C_DIS
LIN {X 111.734,Y 121.731,Z 53.000,A 180.000,B 0.000,C 180.000} C_DIS
LIN {X 111.660,Y 121.567,Z 53.000,A 180.000,B 0.000,C 180.000} C_DIS
LIN {X 111.556,Y 121.325,Z 53.000,A 180.000,B 0.000,C 180.000} C_DIS
LIN {X 111.509,Y 121.209,Z 53.000,A 180.000,B 0.000,C 180.000} C_DIS
LIN {X 111.377,Y 120.841,Z 53.000,A 180.000,B 0.000,C 180.000} C_DIS
LIN {X 111.326,Y 120.673,Z 53.000,A 180.000,B 0.000,C 180.000} C_DIS
LIN {X 111.274,Y 120.494,Z 53.000,A 180.000,B 0.000,C 180.000} C_DIS
LIN {X 111.226,Y 120.315,Z 53.000,A 180.000,B 0.000,C 180.000} C_DIS
LIN {X 111.146,Y 119.958,Z 53.000,A 180.000,B 0.000,C 180.000} C_DIS
LIN {X 111.114,Y 119.779,Z 53.000,A 180.000,B 0.000,C 180.000} C_DIS
LIN {X 111.086,Y 119.600,Z 53.000,A 180.000,B 0.000,C 180.000} C_DIS
LIN {X 111.059,Y 119.422,Z 53.000,A 180.000,B 0.000,C 180.000} C_DIS
LIN {X 111.019,Y 119.006,Z 53.000,A 180.000,B 0.000,C 180.000} C_DIS
LIN {X 111.013,Y 118.885,Z 53.000,A 180.000,B 0.000,C 180.000} C_DIS
LIN {X 111.002,Y 118.528,Z 53.000,A 180.000,B 0.000,C 180.000} C_DIS
LIN {X 111.006,Y 118.349,Z 53.000,A 180.000,B 0.000,C 180.000} C_DIS
LIN {X 111.012,Y 118.170,Z 53.000,A 180.000,B 0.000,C 180.000} C_DIS
LIN {X 111.019,Y 117.994,Z 53.000,A 180.000,B 0.000,C 180.000} C_DIS
LIN {X 111.053,Y 117.634,Z 53.000,A 180.000,B 0.000,C 180.000} C_DIS
LIN {X 111.077,Y 117.455,Z 53.000,A 180.000,B 0.000,C 180.000} C_DIS
LIN {X 111.134,Y 117.098,Z 53.000,A 180.000,B 0.000,C 180.000} C_DIS
LIN {X 111.173,Y 116.919,Z 53.000,A 180.000,B 0.000,C 180.000} C_DIS
LIN {X 111.213,Y 116.740,Z 53.000,A 180.000,B 0.000,C 180.000} C_DIS
LIN {X 111.258,Y 116.561,Z 53.000,A 180.000,B 0.000,C 180.000} C_DIS
LIN {X 111.362,Y 116.204,Z 53.000,A 180.000,B 0.000,C 180.000} C_DIS
LIN {X 111.377,Y 116.159,Z 53.000,A 180.000,B 0.000,C 180.000} C_DIS
LIN {X 111.489,Y 115.846,Z 53.000,A 180.000,B 0.000,C 180.000} C_DIS
LIN {X 111.556,Y 115.675,Z 53.000,A 180.000,B 0.000,C 180.000} C_DIS
LIN {X 111.714,Y 115.310,Z 53.000,A 180.000,B 0.000,C 180.000} C_DIS
LIN {X 111.734,Y 115.269,Z 53.000,A 180.000,B 0.000,C 180.000} C_DIS
LIN {X 111.913,Y 114.918,Z 53.000,A 180.000,B 0.000,C 180.000} C_DIS
LIN {X 111.996,Y 114.774,Z 53.000,A 180.000,B 0.000,C 180.000} C_DIS
LIN {X 112.102,Y 114.595,Z 53.000,A 180.000,B 0.000,C 180.000} C_DIS
LIN {X 112.213,Y 114.416,Z 53.000,A 180.000,B 0.000,C 180.000} C_DIS
LIN {X 112.335,Y 114.237,Z 53.000,A 180.000,B 0.000,C 180.000} C_DIS
LIN {X 112.450,Y 114.072,Z 53.000,A 180.000,B 0.000,C 180.000} C_DIS
LIN {X 112.628,Y 113.841,Z 53.000,A 180.000,B 0.000,C 180.000} C_DIS
LIN {X 112.739,Y 113.701,Z 53.000,A 180.000,B 0.000,C 180.000} C_DIS
LIN {X 112.986,Y 113.421,Z 53.000,A 180.000,B 0.000,C 180.000} C_DIS
LIN {X 113.057,Y 113.343,Z 53.000,A 180.000,B 0.000,C 180.000} C_DIS
LIN {X 113.343,Y 113.057,Z 53.000,A 180.000,B 0.000,C 180.000} C_DIS
LIN {X 113.421,Y 112.986,Z 53.000,A 180.000,B 0.000,C 180.000} C_DIS
LIN {X 113.701,Y 112.739,Z 53.000,A 180.000,B 0.000,C 180.000} C_DIS
LIN {X 113.841,Y 112.628,Z 53.000,A 180.000,B 0.000,C 180.000} C_DIS
LIN {X 114.072,Y 112.450,Z 53.000,A 180.000,B 0.000,C 180.000} C_DIS
LIN {X 114.237,Y 112.335,Z 53.000,A 180.000,B 0.000,C 180.000} C_DIS
LIN {X 114.416,Y 112.213,Z 53.000,A 180.000,B 0.000,C 180.000} C_DIS
LIN {X 114.595,Y 112.102,Z 53.000,A 180.000,B 0.000,C 180.000} C_DIS
LIN {X 114.774,Y 111.996,Z 53.000,A 180.000,B 0.000,C 180.000} C_DIS
LIN {X 114.918,Y 111.913,Z 53.000,A 180.000,B 0.000,C 180.000} C_DIS
LIN {X 115.269,Y 111.734,Z 53.000,A 180.000,B 0.000,C 180.000} C_DIS
LIN {X 115.310,Y 111.714,Z 53.000,A 180.000,B 0.000,C 180.000} C_DIS
LIN {X 115.675,Y 111.556,Z 53.000,A 180.000,B 0.000,C 180.000} C_DIS
LIN {X 115.846,Y 111.489,Z 53.000,A 180.000,B 0.000,C 180.000} C_DIS
LIN {X 116.159,Y 111.377,Z 53.000,A 180.000,B 0.000,C 180.000} C_DIS
LIN {X 116.204,Y 111.362,Z 53.000,A 180.000,B 0.000,C 180.000} C_DIS
LIN {X 116.561,Y 111.258,Z 53.000,A 180.000,B 0.000,C 180.000} C_DIS
LIN {X 116.740,Y 111.213,Z 53.000,A 180.000,B 0.000,C 180.000} C_DIS
LIN {X 116.919,Y 111.173,Z 53.000,A 180.000,B 0.000,C 180.000} C_DIS
LIN {X 117.098,Y 111.134,Z 53.000,A 180.000,B 0.000,C 180.000} C_DIS
LIN {X 117.455,Y 111.077,Z 53.000,A 180.000,B 0.000,C 180.000} C_DIS
LIN {X 117.634,Y 111.053,Z 53.000,A 180.000,B 0.000,C 180.000} C_DIS
LIN {X 117.994,Y 111.019,Z 53.000,A 180.000,B 0.000,C 180.000} C_DIS
LIN {X 118.170,Y 111.012,Z 53.000,A 180.000,B 0.000,C 180.000} C_DIS
LIN {X 118.349,Y 111.006,Z 53.000,A 180.000,B 0.000,C 180.000} C_DIS
LIN {X 118.528,Y 111.002,Z 53.000,A 180.000,B 0.000,C 180.000} C_DIS
LIN {X 118.885,Y 111.013,Z 53.000,A 180.000,B 0.000,C 180.000} C_DIS
LIN {X 119.006,Y 111.019,Z 53.000,A 180.000,B 0.000,C 180.000} C_DIS
LIN {X 119.422,Y 111.059,Z 53.000,A 180.000,B 0.000,C 180.000} C_DIS
LIN {X 119.600,Y 111.086,Z 53.000,A 180.000,B 0.000,C 180.000} C_DIS
LIN {X 119.779,Y 111.114,Z 53.000,A 180.000,B 0.000,C 180.000} C_DIS
LIN {X 119.958,Y 111.146,Z 53.000,A 180.000,B 0.000,C 180.000} C_DIS
LIN {X 120.315,Y 111.226,Z 53.000,A 180.000,B 0.000,C 180.000} C_DIS
LIN {X 120.494,Y 111.274,Z 53.000,A 180.000,B 0.000,C 180.000} C_DIS
LIN {X 120.673,Y 111.326,Z 53.000,A 180.000,B 0.000,C 180.000} C_DIS
LIN {X 120.841,Y 111.377,Z 53.000,A 180.000,B 0.000,C 180.000} C_DIS
LIN {X 121.209,Y 111.509,Z 53.000,A 180.000,B 0.000,C 180.000} C_DIS
LIN {X 121.325,Y 111.556,Z 53.000,A 180.000,B 0.000,C 180.000} C_DIS
LIN {X 121.567,Y 111.660,Z 53.000,A 180.000,B 0.000,C 180.000} C_DIS
LIN {X 121.731,Y 111.734,Z 53.000,A 180.000,B 0.000,C 180.000} C_DIS
LIN {X 122.103,Y 111.924,Z 53.000,A 180.000,B 0.000,C 180.000} C_DIS
LIN {X 122.282,Y 112.029,Z 53.000,A 180.000,B 0.000,C 180.000} C_DIS
LIN {X 122.461,Y 112.135,Z 53.000,A 180.000,B 0.000,C 180.000} C_DIS
LIN {X 122.639,Y 112.251,Z 53.000,A 180.000,B 0.000,C 180.000} C_DIS
LIN {X 122.818,Y 112.373,Z 53.000,A 180.000,B 0.000,C 180.000} C_DIS
LIN {X 122.928,Y 112.450,Z 53.000,A 180.000,B 0.000,C 180.000} C_DIS
LIN {X 123.176,Y 112.641,Z 53.000,A 180.000,B 0.000,C 180.000} C_DIS
LIN {X 123.354,Y 112.788,Z 53.000,A 180.000,B 0.000,C 180.000} C_DIS
LIN {X 123.579,Y 112.986,Z 53.000,A 180.000,B 0.000,C 180.000} C_DIS
LIN {X 123.712,Y 113.112,Z 53.000,A 180.000,B 0.000,C 180.000} C_DIS
LIN {X 123.729,Y 113.130,Z 53.000,A 180.000,B 0.000,C 180.000} C_DIS
; Link Move Starts
LIN {X 123.952,Y 113.352,Z 53.000,A 180.000,B 0.000,C 180.000} C_DIS
LIN {X 124.161,Y 113.588,Z 52.999,A 180.000,B 0.000,C 180.000} C_DIS
LIN {X 124.363,Y 113.830,Z 52.998,A 180.000,B 0.000,C 180.000} C_DIS
LIN {X 124.556,Y 114.079,Z 52.996,A 180.000,B 0.000,C 180.000} C_DIS
LIN {X 124.734,Y 114.339,Z 52.994,A 180.000,B 0.000,C 180.000} C_DIS
LIN {X 124.904,Y 114.604,Z 52.991,A 180.000,B 0.000,C 180.000} C_DIS
LIN {X 125.064,Y 114.875,Z 52.988,A 180.000,B 0.000,C 180.000} C_DIS
LIN {X 125.208,Y 115.155,Z 52.985,A 180.000,B 0.000,C 180.000} C_DIS
LIN {X 125.343,Y 115.440,Z 52.981,A 180.000,B 0.000,C 180.000} C_DIS
LIN {X 125.468,Y 115.729,Z 52.977,A 180.000,B 0.000,C 180.000} C_DIS
LIN {X 125.575,Y 116.025,Z 52.972,A 180.000,B 0.000,C 180.000} C_DIS
LIN {X 125.628,Y 116.173,Z 52.969,A 180.000,B 0.000,C 180.000} C_DIS
LIN {X 125.673,Y 116.324,Z 52.967,A 180.000,B 0.000,C 180.000} C_DIS
LIN {X 125.717,Y 116.476,Z 52.964,A 180.000,B 0.000,C 180.000} C_DIS
LIN {X 125.761,Y 116.627,Z 52.961,A 180.000,B 0.000,C 180.000} C_DIS
LIN {X 125.796,Y 116.781,Z 52.959,A 180.000,B 0.000,C 180.000} C_DIS
LIN {X 125.830,Y 116.934,Z 52.956,A 180.000,B 0.000,C 180.000} C_DIS
LIN {X 125.864,Y 117.088,Z 52.952,A 180.000,B 0.000,C 180.000} C_DIS
LIN {X 125.889,Y 117.244,Z 52.949,A 180.000,B 0.000,C 180.000} C_DIS
LIN {X 125.914,Y 117.399,Z 52.946,A 180.000,B 0.000,C 180.000} C_DIS
LIN {X 125.939,Y 117.555,Z 52.943,A 180.000,B 0.000,C 180.000} C_DIS
LIN {X 125.954,Y 117.711,Z 52.939,A 180.000,B 0.000,C 180.000} C_DIS
LIN {X 125.969,Y 117.868,Z 52.936,A 180.000,B 0.000,C 180.000} C_DIS
LIN {X 125.984,Y 118.025,Z 52.932,A 180.000,B 0.000,C 180.000} C_DIS
LIN {X 125.989,Y 118.183,Z 52.928,A 180.000,B 0.000,C 180.000} C_DIS
LIN {X 125.994,Y 118.340,Z 52.925,A 180.000,B 0.000,C 180.000} C_DIS
LIN {X 125.999,Y 118.497,Z 52.921,A 180.000,B 0.000,C 180.000} C_DIS
LIN {X 125.994,Y 118.655,Z 52.917,A 180.000,B 0.000,C 180.000} C_DIS
LIN {X 125.989,Y 118.812,Z 52.913,A 180.000,B 0.000,C 180.000} C_DIS
LIN {X 125.984,Y 118.970,Z 52.909,A 180.000,B 0.000,C 180.000} C_DIS
LIN {X 125.969,Y 119.127,Z 52.905,A 180.000,B 0.000,C 180.000} C_DIS
LIN {X 125.954,Y 119.283,Z 52.900,A 180.000,B 0.000,C 180.000} C_DIS
LIN {X 125.940,Y 119.440,Z 52.896,A 180.000,B 0.000,C 180.000} C_DIS
LIN {X 125.915,Y 119.596,Z 52.892,A 180.000,B 0.000,C 180.000} C_DIS
LIN {X 125.890,Y 119.751,Z 52.887,A 180.000,B 0.000,C 180.000} C_DIS
LIN {X 125.866,Y 119.907,Z 52.883,A 180.000,B 0.000,C 180.000} C_DIS
LIN {X 125.831,Y 120.061,Z 52.878,A 180.000,B 0.000,C 180.000} C_DIS
LIN {X 125.797,Y 120.214,Z 52.873,A 180.000,B 0.000,C 180.000} C_DIS
LIN {X 125.762,Y 120.368,Z 52.869,A 180.000,B 0.000,C 180.000} C_DIS
LIN {X 125.718,Y 120.519,Z 52.864,A 180.000,B 0.000,C 180.000} C_DIS
LIN {X 125.674,Y 120.671,Z 52.859,A 180.000,B 0.000,C 180.000} C_DIS
LIN {X 125.630,Y 120.822,Z 52.854,A 180.000,B 0.000,C 180.000} C_DIS
LIN {X 125.603,Y 120.896,Z 52.851,A 180.000,B 0.000,C 180.000} C_DIS
LIN {X 125.577,Y 120.970,Z 52.849,A 180.000,B 0.000,C 180.000} C_DIS
LIN {X 125.550,Y 121.044,Z 52.846,A 180.000,B 0.000,C 180.000} C_DIS
LIN {X 125.523,Y 121.118,Z 52.844,A 180.000,B 0.000,C 180.000} C_DIS
LIN {X 125.497,Y 121.192,Z 52.841,A 180.000,B 0.000,C 180.000} C_DIS
LIN {X 125.470,Y 121.266,Z 52.839,A 180.000,B 0.000,C 180.000} C_DIS
LIN {X 125.438,Y 121.339,Z 52.836,A 180.000,B 0.000,C 180.000} C_DIS
LIN {X 125.376,Y 121.483,Z 52.831,A 180.000,B 0.000,C 180.000} C_DIS
LIN {X 125.313,Y 121.628,Z 52.825,A 180.000,B 0.000,C 180.000} C_DIS
LIN {X 125.282,Y 121.700,Z 52.823,A 180.000,B 0.000,C 180.000} C_DIS
LIN {X 125.210,Y 121.840,Z 52.817,A 180.000,B 0.000,C 180.000} C_DIS
LIN {X 125.139,Y 121.980,Z 52.812,A 180.000,B 0.000,C 180.000} C_DIS
LIN {X 125.103,Y 122.051,Z 52.809,A 180.000,B 0.000,C 180.000} C_DIS
LIN {X 125.067,Y 122.120,Z 52.806,A 180.000,B 0.000,C 180.000} C_DIS
LIN {X 124.986,Y 122.256,Z 52.801,A 180.000,B 0.000,C 180.000} C_DIS
LIN {X 124.866,Y 122.459,Z 52.793,A 180.000,B 0.000,C 180.000} C_DIS
LIN {X 124.825,Y 122.527,Z 52.790,A 180.000,B 0.000,C 180.000} C_DIS
LIN {X 124.693,Y 122.722,Z 52.782,A 180.000,B 0.000,C 180.000} C_DIS
LIN {X 124.604,Y 122.853,Z 52.776,A 180.000,B 0.000,C 180.000} C_DIS
LIN {X 124.559,Y 122.917,Z 52.774,A 180.000,B 0.000,C 180.000} C_DIS
LIN {X 124.463,Y 123.042,Z 52.768,A 180.000,B 0.000,C 180.000} C_DIS
LIN {X 124.318,Y 123.228,Z 52.760,A 180.000,B 0.000,C 180.000} C_DIS
LIN {X 124.269,Y 123.290,Z 52.757,A 180.000,B 0.000,C 180.000} C_DIS
LIN {X 124.113,Y 123.467,Z 52.749,A 180.000,B 0.000,C 180.000} C_DIS
LIN {X 124.008,Y 123.586,Z 52.743,A 180.000,B 0.000,C 180.000} C_DIS
LIN {X 123.956,Y 123.644,Z 52.741,A 180.000,B 0.000,C 180.000} C_DIS
LIN {X 123.844,Y 123.755,Z 52.735,A 180.000,B 0.000,C 180.000} C_DIS
LIN {X 123.677,Y 123.922,Z 52.727,A 180.000,B 0.000,C 180.000} C_DIS
LIN {X 123.621,Y 123.977,Z 52.724,A 180.000,B 0.000,C 180.000} C_DIS
LIN {X 123.325,Y 124.238,Z 52.710,A 180.000,B 0.000,C 180.000} C_DIS
LIN {X 123.266,Y 124.289,Z 52.708,A 180.000,B 0.000,C 180.000} C_DIS
LIN {X 123.141,Y 124.386,Z 52.702,A 180.000,B 0.000,C 180.000} C_DIS
LIN {X 122.954,Y 124.530,Z 52.694,A 180.000,B 0.000,C 180.000} C_DIS
LIN {X 122.891,Y 124.578,Z 52.691,A 180.000,B 0.000,C 180.000} C_DIS
LIN {X 122.566,Y 124.799,Z 52.677,A 180.000,B 0.000,C 180.000} C_DIS
LIN {X 122.500,Y 124.842,Z 52.675,A 180.000,B 0.000,C 180.000} C_DIS
LIN {X 122.364,Y 124.922,Z 52.669,A 180.000,B 0.000,C 180.000} C_DIS
LIN {X 122.161,Y 125.043,Z 52.661,A 180.000,B 0.000,C 180.000} C_DIS
LIN {X 122.092,Y 125.082,Z 52.658,A 180.000,B 0.000,C 180.000} C_DIS
LIN {X 121.742,Y 125.260,Z 52.644,A 180.000,B 0.000,C 180.000} C_DIS
LIN {X 121.671,Y 125.295,Z 52.642,A 180.000,B 0.000,C 180.000} C_DIS
LIN {X 121.454,Y 125.388,Z 52.633,A 180.000,B 0.000,C 180.000} C_DIS
LIN {X 121.309,Y 125.451,Z 52.628,A 180.000,B 0.000,C 180.000} C_DIS
LIN {X 121.236,Y 125.481,Z 52.625,A 180.000,B 0.000,C 180.000} C_DIS
LIN {X 120.866,Y 125.614,Z 52.611,A 180.000,B 0.000,C 180.000} C_DIS
LIN {X 120.791,Y 125.639,Z 52.609,A 180.000,B 0.000,C 180.000} C_DIS
LIN {X 120.564,Y 125.705,Z 52.600,A 180.000,B 0.000,C 180.000} C_DIS
LIN {X 120.413,Y 125.749,Z 52.595,A 180.000,B 0.000,C 180.000} C_DIS
LIN {X 120.337,Y 125.769,Z 52.592,A 180.000,B 0.000,C 180.000} C_DIS
LIN {X 119.953,Y 125.855,Z 52.578,A 180.000,B 0.000,C 180.000} C_DIS
LIN {X 119.875,Y 125.871,Z 52.576,A 180.000,B 0.000,C 180.000} C_DIS
LIN {X 119.487,Y 125.932,Z 52.562,A 180.000,B 0.000,C 180.000} C_DIS
LIN {X 119.408,Y 125.943,Z 52.559,A 180.000,B 0.000,C 180.000} C_DIS
LIN {X 119.016,Y 125.980,Z 52.545,A 180.000,B 0.000,C 180.000} C_DIS
LIN {X 118.938,Y 125.985,Z 52.543,A 180.000,B 0.000,C 180.000} C_DIS
LIN {X 118.544,Y 125.997,Z 52.529,A 180.000,B 0.000,C 180.000} C_DIS
LIN {X 118.466,Y 125.998,Z 52.526,A 180.000,B 0.000,C 180.000} C_DIS
LIN {X 118.072,Y 125.985,Z 52.512,A 180.000,B 0.000,C 180.000} C_DIS
LIN {X 117.993,Y 125.981,Z 52.510,A 180.000,B 0.000,C 180.000} C_DIS
LIN {X 117.601,Y 125.944,Z 52.496,A 180.000,B 0.000,C 180.000} C_DIS
LIN {X 117.523,Y 125.934,Z 52.493,A 180.000,B 0.000,C 180.000} C_DIS
LIN {X 117.134,Y 125.872,Z 52.479,A 180.000,B 0.000,C 180.000} C_DIS
LIN {X 117.057,Y 125.857,Z 52.477,A 180.000,B 0.000,C 180.000} C_DIS
LIN {X 116.673,Y 125.772,Z 52.463,A 180.000,B 0.000,C 180.000} C_DIS
LIN {X 116.596,Y 125.752,Z 52.460,A 180.000,B 0.000,C 180.000} C_DIS
LIN {X 116.218,Y 125.642,Z 52.446,A 180.000,B 0.000,C 180.000} C_DIS
LIN {X 116.143,Y 125.618,Z 52.444,A 180.000,B 0.000,C 180.000} C_DIS
LIN {X 115.773,Y 125.484,Z 52.430,A 180.000,B 0.000,C 180.000} C_DIS
LIN {X 115.700,Y 125.455,Z 52.427,A 180.000,B 0.000,C 180.000} C_DIS
LIN {X 115.338,Y 125.299,Z 52.413,A 180.000,B 0.000,C 180.000} C_DIS
LIN {X 115.267,Y 125.265,Z 52.411,A 180.000,B 0.000,C 180.000} C_DIS
LIN {X 115.057,Y 125.158,Z 52.402,A 180.000,B 0.000,C 180.000} C_DIS
LIN {X 114.916,Y 125.086,Z 52.397,A 180.000,B 0.000,C 180.000} C_DIS
LIN {X 114.848,Y 125.048,Z 52.394,A 180.000,B 0.000,C 180.000} C_DIS
LIN {X 114.509,Y 124.847,Z 52.380,A 180.000,B 0.000,C 180.000} C_DIS
LIN {X 114.442,Y 124.805,Z 52.378,A 180.000,B 0.000,C 180.000} C_DIS
LIN {X 114.247,Y 124.672,Z 52.369,A 180.000,B 0.000,C 180.000} C_DIS
LIN {X 114.117,Y 124.583,Z 52.364,A 180.000,B 0.000,C 180.000} C_DIS
LIN {X 114.053,Y 124.536,Z 52.361,A 180.000,B 0.000,C 180.000} C_DIS
LIN {X 113.742,Y 124.295,Z 52.347,A 180.000,B 0.000,C 180.000} C_DIS
LIN {X 113.682,Y 124.244,Z 52.345,A 180.000,B 0.000,C 180.000} C_DIS
LIN {X 113.505,Y 124.088,Z 52.336,A 180.000,B 0.000,C 180.000} C_DIS
LIN {X 113.387,Y 123.984,Z 52.331,A 180.000,B 0.000,C 180.000} C_DIS
LIN {X 113.330,Y 123.929,Z 52.328,A 180.000,B 0.000,C 180.000} C_DIS
LIN {X 113.051,Y 123.651,Z 52.314,A 180.000,B 0.000,C 180.000} C_DIS
LIN {X 112.998,Y 123.593,Z 52.312,A 180.000,B 0.000,C 180.000} C_DIS
LIN {X 112.894,Y 123.475,Z 52.306,A 180.000,B 0.000,C 180.000} C_DIS
LIN {X 112.738,Y 123.298,Z 52.298,A 180.000,B 0.000,C 180.000} C_DIS
LIN {X 112.688,Y 123.236,Z 52.295,A 180.000,B 0.000,C 180.000} C_DIS
LIN {X 112.543,Y 123.050,Z 52.287,A 180.000,B 0.000,C 180.000} C_DIS
LIN {X 112.447,Y 122.925,Z 52.281,A 180.000,B 0.000,C 180.000} C_DIS
LIN {X 112.402,Y 122.861,Z 52.279,A 180.000,B 0.000,C 180.000} C_DIS
LIN {X 112.313,Y 122.731,Z 52.273,A 180.000,B 0.000,C 180.000} C_DIS
LIN {X 112.180,Y 122.535,Z 52.265,A 180.000,B 0.000,C 180.000} C_DIS
LIN {X 112.139,Y 122.468,Z 52.262,A 180.000,B 0.000,C 180.000} C_DIS
LIN {X 112.019,Y 122.265,Z 52.254,A 180.000,B 0.000,C 180.000} C_DIS
LIN {X 111.939,Y 122.129,Z 52.248,A 180.000,B 0.000,C 180.000} C_DIS
LIN {X 111.902,Y 122.059,Z 52.246,A 180.000,B 0.000,C 180.000} C_DIS
LIN {X 111.830,Y 121.919,Z 52.240,A 180.000,B 0.000,C 180.000} C_DIS
LIN {X 111.723,Y 121.709,Z 52.232,A 180.000,B 0.000,C 180.000} C_DIS
LIN {X 111.691,Y 121.637,Z 52.229,A 180.000,B 0.000,C 180.000} C_DIS
LIN {X 111.597,Y 121.420,Z 52.221,A 180.000,B 0.000,C 180.000} C_DIS
LIN {X 111.534,Y 121.275,Z 52.215,A 180.000,B 0.000,C 180.000} C_DIS
LIN {X 111.507,Y 121.202,Z 52.213,A 180.000,B 0.000,C 180.000} C_DIS
LIN {X 111.453,Y 121.053,Z 52.207,A 180.000,B 0.000,C 180.000} C_DIS
LIN {X 111.373,Y 120.831,Z 52.199,A 180.000,B 0.000,C 180.000} C_DIS
LIN {X 111.350,Y 120.756,Z 52.196,A 180.000,B 0.000,C 180.000} C_DIS
LIN {X 111.306,Y 120.605,Z 52.191,A 180.000,B 0.000,C 180.000} C_DIS
LIN {X 111.263,Y 120.453,Z 52.185,A 180.000,B 0.000,C 180.000} C_DIS
LIN {X 111.241,Y 120.378,Z 52.182,A 180.000,B 0.000,C 180.000} C_DIS
LIN {X 111.223,Y 120.301,Z 52.180,A 180.000,B 0.000,C 180.000} C_DIS
LIN {X 111.188,Y 120.147,Z 52.174,A 180.000,B 0.000,C 180.000} C_DIS
LIN {X 111.154,Y 119.994,Z 52.169,A 180.000,B 0.000,C 180.000} C_DIS
LIN {X 111.137,Y 119.917,Z 52.166,A 180.000,B 0.000,C 180.000} C_DIS
LIN {X 111.124,Y 119.839,Z 52.164,A 180.000,B 0.000,C 180.000} C_DIS
LIN {X 111.111,Y 119.761,Z 52.161,A 180.000,B 0.000,C 180.000} C_DIS
LIN {X 111.099,Y 119.683,Z 52.159,A 180.000,B 0.000,C 180.000} C_DIS
LIN {X 111.087,Y 119.606,Z 52.156,A 180.000,B 0.000,C 180.000} C_DIS
LIN {X 111.074,Y 119.528,Z 52.154,A 180.000,B 0.000,C 180.000} C_DIS
LIN {X 111.062,Y 119.450,Z 52.151,A 180.000,B 0.000,C 180.000} C_DIS
LIN {X 111.054,Y 119.372,Z 52.149,A 180.000,B 0.000,C 180.000} C_DIS
LIN {X 111.039,Y 119.215,Z 52.144,A 180.000,B 0.000,C 180.000} C_DIS
LIN {X 111.024,Y 119.058,Z 52.139,A 180.000,B 0.000,C 180.000} C_DIS
LIN {X 111.014,Y 118.901,Z 52.134,A 180.000,B 0.000,C 180.000} C_DIS
LIN {X 111.009,Y 118.744,Z 52.129,A 180.000,B 0.000,C 180.000} C_DIS
LIN {X 111.004,Y 118.586,Z 52.124,A 180.000,B 0.000,C 180.000} C_DIS
LIN {X 111.003,Y 118.429,Z 52.120,A 180.000,B 0.000,C 180.000} C_DIS
LIN {X 111.008,Y 118.271,Z 52.115,A 180.000,B 0.000,C 180.000} C_DIS
LIN {X 111.013,Y 118.114,Z 52.111,A 180.000,B 0.000,C 180.000} C_DIS
LIN {X 111.023,Y 117.957,Z 52.106,A 180.000,B 0.000,C 180.000} C_DIS
LIN {X 111.038,Y 117.800,Z 52.102,A 180.000,B 0.000,C 180.000} C_DIS
LIN {X 111.053,Y 117.643,Z 52.097,A 180.000,B 0.000,C 180.000} C_DIS
LIN {X 111.072,Y 117.487,Z 52.093,A 180.000,B 0.000,C 180.000} C_DIS
LIN {X 111.097,Y 117.331,Z 52.089,A 180.000,B 0.000,C 180.000} C_DIS
LIN {X 111.121,Y 117.176,Z 52.085,A 180.000,B 0.000,C 180.000} C_DIS
LIN {X 111.151,Y 117.021,Z 52.081,A 180.000,B 0.000,C 180.000} C_DIS
LIN {X 111.185,Y 116.867,Z 52.077,A 180.000,B 0.000,C 180.000} C_DIS
LIN {X 111.219,Y 116.714,Z 52.073,A 180.000,B 0.000,C 180.000} C_DIS
LIN {X 111.258,Y 116.561,Z 52.070,A 180.000,B 0.000,C 180.000} C_DIS
LIN {X 111.302,Y 116.410,Z 52.066,A 180.000,B 0.000,C 180.000} C_DIS
LIN {X 111.346,Y 116.258,Z 52.062,A 180.000,B 0.000,C 180.000} C_DIS
LIN {X 111.395,Y 116.109,Z 52.059,A 180.000,B 0.000,C 180.000} C_DIS
LIN {X 111.448,Y 115.961,Z 52.056,A 180.000,B 0.000,C 180.000} C_DIS
LIN {X 111.502,Y 115.812,Z 52.052,A 180.000,B 0.000,C 180.000} C_DIS
LIN {X 111.560,Y 115.666,Z 52.049,A 180.000,B 0.000,C 180.000} C_DIS
LIN {X 111.622,Y 115.521,Z 52.046,A 180.000,B 0.000,C 180.000} C_DIS
LIN {X 111.685,Y 115.377,Z 52.043,A 180.000,B 0.000,C 180.000} C_DIS
LIN {X 111.752,Y 115.234,Z 52.040,A 180.000,B 0.000,C 180.000} C_DIS
LIN {X 111.823,Y 115.094,Z 52.037,A 180.000,B 0.000,C 180.000} C_DIS
LIN {X 111.895,Y 114.954,Z 52.034,A 180.000,B 0.000,C 180.000} C_DIS
LIN {X 111.971,Y 114.816,Z 52.032,A 180.000,B 0.000,C 180.000} C_DIS
LIN {X 112.051,Y 114.680,Z 52.029,A 180.000,B 0.000,C 180.000} C_DIS
LIN {X 112.131,Y 114.545,Z 52.027,A 180.000,B 0.000,C 180.000} C_DIS
LIN {X 112.305,Y 114.282,Z 52.022,A 180.000,B 0.000,C 180.000} C_DIS
LIN {X 112.486,Y 114.024,Z 52.018,A 180.000,B 0.000,C 180.000} C_DIS
LIN {X 112.679,Y 113.775,Z 52.014,A 180.000,B 0.000,C 180.000} C_DIS
LIN {X 112.884,Y 113.536,Z 52.011,A 180.000,B 0.000,C 180.000} C_DIS
LIN {X 113.097,Y 113.304,Z 52.008,A 180.000,B 0.000,C 180.000} C_DIS
LIN {X 113.319,Y 113.081,Z 52.005,A 180.000,B 0.000,C 180.000} C_DIS
LIN {X 113.553,Y 112.870,Z 52.003,A 180.000,B 0.000,C 180.000} C_DIS
LIN {X 113.793,Y 112.666,Z 52.002,A 180.000,B 0.000,C 180.000} C_DIS
LIN {X 114.042,Y 112.473,Z 52.001,A 180.000,B 0.000,C 180.000} C_DIS
LIN {X 114.300,Y 112.292,Z 52.000,A 180.000,B 0.000,C 180.000} C_DIS
LIN {X 114.494,Y 112.165,Z 52.000,A 180.000,B 0.000,C 180.000} C_DIS
; Cutting Move Starts
LIN {X 114.595,Y 112.102,Z 52.000,A 180.000,B 0.000,C 180.000} C_DIS
LIN {X 114.774,Y 111.996,Z 52.000,A 180.000,B 0.000,C 180.000} C_DIS
LIN {X 114.918,Y 111.913,Z 52.000,A 180.000,B 0.000,C 180.000} C_DIS
LIN {X 115.269,Y 111.734,Z 52.000,A 180.000,B 0.000,C 180.000} C_DIS
LIN {X 115.310,Y 111.714,Z 52.000,A 180.000,B 0.000,C 180.000} C_DIS
LIN {X 115.675,Y 111.556,Z 52.000,A 180.000,B 0.000,C 180.000} C_DIS
LIN {X 115.846,Y 111.489,Z 52.000,A 180.000,B 0.000,C 180.000} C_DIS
LIN {X 116.159,Y 111.377,Z 52.000,A 180.000,B 0.000,C 180.000} C_DIS
LIN {X 116.204,Y 111.362,Z 52.000,A 180.000,B 0.000,C 180.000} C_DIS
LIN {X 116.561,Y 111.258,Z 52.000,A 180.000,B 0.000,C 180.000} C_DIS
LIN {X 116.740,Y 111.213,Z 52.000,A 180.000,B 0.000,C 180.000} C_DIS
LIN {X 116.919,Y 111.173,Z 52.000,A 180.000,B 0.000,C 180.000} C_DIS
LIN {X 117.098,Y 111.134,Z 52.000,A 180.000,B 0.000,C 180.000} C_DIS
LIN {X 117.455,Y 111.077,Z 52.000,A 180.000,B 0.000,C 180.000} C_DIS
LIN {X 117.634,Y 111.053,Z 52.000,A 180.000,B 0.000,C 180.000} C_DIS
LIN {X 117.994,Y 111.019,Z 52.000,A 180.000,B 0.000,C 180.000} C_DIS
LIN {X 118.170,Y 111.012,Z 52.000,A 180.000,B 0.000,C 180.000} C_DIS
LIN {X 118.349,Y 111.006,Z 52.000,A 180.000,B 0.000,C 180.000} C_DIS
LIN {X 118.528,Y 111.002,Z 52.000,A 180.000,B 0.000,C 180.000} C_DIS
LIN {X 118.885,Y 111.013,Z 52.000,A 180.000,B 0.000,C 180.000} C_DIS
LIN {X 119.006,Y 111.019,Z 52.000,A 180.000,B 0.000,C 180.000} C_DIS
LIN {X 119.422,Y 111.059,Z 52.000,A 180.000,B 0.000,C 180.000} C_DIS
LIN {X 119.600,Y 111.086,Z 52.000,A 180.000,B 0.000,C 180.000} C_DIS
LIN {X 119.779,Y 111.114,Z 52.000,A 180.000,B 0.000,C 180.000} C_DIS
LIN {X 119.958,Y 111.146,Z 52.000,A 180.000,B 0.000,C 180.000} C_DIS
LIN {X 120.315,Y 111.226,Z 52.000,A 180.000,B 0.000,C 180.000} C_DIS
LIN {X 120.494,Y 111.274,Z 52.000,A 180.000,B 0.000,C 180.000} C_DIS
LIN {X 120.673,Y 111.326,Z 52.000,A 180.000,B 0.000,C 180.000} C_DIS
LIN {X 120.841,Y 111.377,Z 52.000,A 180.000,B 0.000,C 180.000} C_DIS
LIN {X 121.209,Y 111.509,Z 52.000,A 180.000,B 0.000,C 180.000} C_DIS
LIN {X 121.325,Y 111.556,Z 52.000,A 180.000,B 0.000,C 180.000} C_DIS
LIN {X 121.567,Y 111.660,Z 52.000,A 180.000,B 0.000,C 180.000} C_DIS
LIN {X 121.731,Y 111.734,Z 52.000,A 180.000,B 0.000,C 180.000} C_DIS
LIN {X 122.103,Y 111.924,Z 52.000,A 180.000,B 0.000,C 180.000} C_DIS
LIN {X 122.282,Y 112.029,Z 52.000,A 180.000,B 0.000,C 180.000} C_DIS
LIN {X 122.461,Y 112.135,Z 52.000,A 180.000,B 0.000,C 180.000} C_DIS
LIN {X 122.639,Y 112.251,Z 52.000,A 180.000,B 0.000,C 180.000} C_DIS
LIN {X 122.818,Y 112.373,Z 52.000,A 180.000,B 0.000,C 180.000} C_DIS
LIN {X 122.928,Y 112.450,Z 52.000,A 180.000,B 0.000,C 180.000} C_DIS
LIN {X 123.176,Y 112.641,Z 52.000,A 180.000,B 0.000,C 180.000} C_DIS
LIN {X 123.354,Y 112.788,Z 52.000,A 180.000,B 0.000,C 180.000} C_DIS
LIN {X 123.579,Y 112.986,Z 52.000,A 180.000,B 0.000,C 180.000} C_DIS
LIN {X 123.712,Y 113.112,Z 52.000,A 180.000,B 0.000,C 180.000} C_DIS
LIN {X 123.943,Y 113.343,Z 52.000,A 180.000,B 0.000,C 180.000} C_DIS
LIN {X 124.070,Y 113.484,Z 52.000,A 180.000,B 0.000,C 180.000} C_DIS
LIN {X 124.261,Y 113.701,Z 52.000,A 180.000,B 0.000,C 180.000} C_DIS
LIN {X 124.402,Y 113.880,Z 52.000,A 180.000,B 0.000,C 180.000} C_DIS
LIN {X 124.540,Y 114.058,Z 52.000,A 180.000,B 0.000,C 180.000} C_DIS
LIN {X 124.606,Y 114.150,Z 52.000,A 180.000,B 0.000,C 180.000} C_DIS
LIN {X 124.787,Y 114.416,Z 52.000,A 180.000,B 0.000,C 180.000} C_DIS
LIN {X 124.898,Y 114.595,Z 52.000,A 180.000,B 0.000,C 180.000} C_DIS
LIN {X 125.004,Y 114.774,Z 52.000,A 180.000,B 0.000,C 180.000} C_DIS
LIN {X 125.104,Y 114.952,Z 52.000,A 180.000,B 0.000,C 180.000} C_DIS
LIN {X 125.195,Y 115.131,Z 52.000,A 180.000,B 0.000,C 180.000} C_DIS
LIN {X 125.286,Y 115.310,Z 52.000,A 180.000,B 0.000,C 180.000} C_DIS
LIN {X 125.441,Y 115.667,Z 52.000,A 180.000,B 0.000,C 180.000} C_DIS
LIN {X 125.500,Y 115.816,Z 52.000,A 180.000,B 0.000,C 180.000} C_DIS
LIN {X 125.575,Y 116.025,Z 52.000,A 180.000,B 0.000,C 180.000} C_DIS
LIN {X 125.638,Y 116.204,Z 52.000,A 180.000,B 0.000,C 180.000} C_DIS
LIN {X 125.742,Y 116.561,Z 52.000,A 180.000,B 0.000,C 180.000} C_DIS
LIN {X 125.787,Y 116.740,Z 52.000,A 180.000,B 0.000,C 180.000} C_DIS
LIN {X 125.857,Y 117.056,Z 52.000,A 180.000,B 0.000,C 180.000} C_DIS
LIN {X 125.866,Y 117.098,Z 52.000,A 180.000,B 0.000,C 180.000} C_DIS
LIN {X 125.923,Y 117.455,Z 52.000,A 180.000,B 0.000,C 180.000} C_DIS
LIN {X 125.947,Y 117.634,Z 52.000,A 180.000,B 0.000,C 180.000} C_DIS
LIN {X 125.980,Y 117.991,Z 52.000,A 180.000,B 0.000,C 180.000} C_DIS
LIN {X 125.988,Y 118.170,Z 52.000,A 180.000,B 0.000,C 180.000} C_DIS
LIN {X 125.994,Y 118.349,Z 52.000,A 180.000,B 0.000,C 180.000} C_DIS
LIN {X 125.998,Y 118.528,Z 52.000,A 180.000,B 0.000,C 180.000} C_DIS
LIN {X 125.987,Y 118.885,Z 52.000,A 180.000,B 0.000,C 180.000} C_DIS
LIN {X 125.975,Y 119.064,Z 52.000,A 180.000,B 0.000,C 180.000} C_DIS
LIN {X 125.941,Y 119.422,Z 52.000,A 180.000,B 0.000,C 180.000} C_DIS
LIN {X 125.914,Y 119.600,Z 52.000,A 180.000,B 0.000,C 180.000} C_DIS
LIN {X 125.886,Y 119.779,Z 52.000,A 180.000,B 0.000,C 180.000} C_DIS
LIN {X 125.857,Y 119.944,Z 52.000,A 180.000,B 0.000,C 180.000} C_DIS
LIN {X 125.774,Y 120.315,Z 52.000,A 180.000,B 0.000,C 180.000} C_DIS
LIN {X 125.726,Y 120.494,Z 52.000,A 180.000,B 0.000,C 180.000} C_DIS
LIN {X 125.674,Y 120.673,Z 52.000,A 180.000,B 0.000,C 180.000} C_DIS
LIN {X 125.619,Y 120.852,Z 52.000,A 180.000,B 0.000,C 180.000} C_DIS
LIN {X 125.491,Y 121.209,Z 52.000,A 180.000,B 0.000,C 180.000} C_DIS
LIN {X 125.417,Y 121.388,Z 52.000,A 180.000,B 0.000,C 180.000} C_DIS
LIN {X 125.321,Y 121.610,Z 52.000,A 180.000,B 0.000,C 180.000} C_DIS
LIN {X 125.258,Y 121.746,Z 52.000,A 180.000,B 0.000,C 180.000} C_DIS
LIN {X 125.076,Y 122.103,Z 52.000,A 180.000,B 0.000,C 180.000} C_DIS
LIN {X 124.971,Y 122.282,Z 52.000,A 180.000,B 0.000,C 180.000} C_DIS
LIN {X 124.865,Y 122.461,Z 52.000,A 180.000,B 0.000,C 180.000} C_DIS
LIN {X 124.785,Y 122.587,Z 52.000,A 180.000,B 0.000,C 180.000} C_DIS
LIN {X 124.606,Y 122.850,Z 52.000,A 180.000,B 0.000,C 180.000} C_DIS
LIN {X 124.497,Y 122.997,Z 52.000,A 180.000,B 0.000,C 180.000} C_DIS
LIN {X 124.359,Y 123.176,Z 52.000,A 180.000,B 0.000,C 180.000} C_DIS
LIN {X 124.248,Y 123.313,Z 52.000,A 180.000,B 0.000,C 180.000} C_DIS
LIN {X 124.055,Y 123.533,Z 52.000,A 180.000,B 0.000,C 180.000} C_DIS
LIN {X 123.891,Y 123.709,Z 52.000,A 180.000,B 0.000,C 180.000} C_DIS
LIN {X 123.709,Y 123.891,Z 52.000,A 180.000,B 0.000,C 180.000} C_DIS
LIN {X 123.533,Y 124.055,Z 52.000,A 180.000,B 0.000,C 180.000} C_DIS
LIN {X 123.313,Y 124.248,Z 52.000,A 180.000,B 0.000,C 180.000} C_DIS
LIN {X 123.176,Y 124.359,Z 52.000,A 180.000,B 0.000,C 180.000} C_DIS
LIN {X 122.997,Y 124.497,Z 52.000,A 180.000,B 0.000,C 180.000} C_DIS
LIN {X 122.850,Y 124.606,Z 52.000,A 180.000,B 0.000,C 180.000} C_DIS
LIN {X 122.587,Y 124.785,Z 52.000,A 180.000,B 0.000,C 180.000} C_DIS
LIN {X 122.461,Y 124.865,Z 52.000,A 180.000,B 0.000,C 180.000} C_DIS
LIN {X 122.282,Y 124.971,Z 52.000,A 180.000,B 0.000,C 180.000} C_DIS
LIN {X 122.103,Y 125.076,Z 52.000,A 180.000,B 0.000,C 180.000} C_DIS
LIN {X 121.746,Y 125.258,Z 52.000,A 180.000,B 0.000,C 180.000} C_DIS
LIN {X 121.610,Y 125.321,Z 52.000,A 180.000,B 0.000,C 180.000} C_DIS
LIN {X 121.388,Y 125.417,Z 52.000,A 180.000,B 0.000,C 180.000} C_DIS
LIN {X 121.209,Y 125.491,Z 52.000,A 180.000,B 0.000,C 180.000} C_DIS
LIN {X 120.852,Y 125.619,Z 52.000,A 180.000,B 0.000,C 180.000} C_DIS
LIN {X 120.673,Y 125.674,Z 52.000,A 180.000,B 0.000,C 180.000} C_DIS
LIN {X 120.494,Y 125.726,Z 52.000,A 180.000,B 0.000,C 180.000} C_DIS
LIN {X 120.315,Y 125.774,Z 52.000,A 180.000,B 0.000,C 180.000} C_DIS
LIN {X 119.944,Y 125.857,Z 52.000,A 180.000,B 0.000,C 180.000} C_DIS
LIN {X 119.779,Y 125.886,Z 52.000,A 180.000,B 0.000,C 180.000} C_DIS
LIN {X 119.600,Y 125.914,Z 52.000,A 180.000,B 0.000,C 180.000} C_DIS
LIN {X 119.422,Y 125.941,Z 52.000,A 180.000,B 0.000,C 180.000} C_DIS
LIN {X 119.064,Y 125.975,Z 52.000,A 180.000,B 0.000,C 180.000} C_DIS
LIN {X 118.885,Y 125.987,Z 52.000,A 180.000,B 0.000,C 180.000} C_DIS
LIN {X 118.528,Y 125.998,Z 52.000,A 180.000,B 0.000,C 180.000} C_DIS
LIN {X 118.349,Y 125.994,Z 52.000,A 180.000,B 0.000,C 180.000} C_DIS
LIN {X 118.170,Y 125.988,Z 52.000,A 180.000,B 0.000,C 180.000} C_DIS
LIN {X 117.991,Y 125.980,Z 52.000,A 180.000,B 0.000,C 180.000} C_DIS
LIN {X 117.634,Y 125.947,Z 52.000,A 180.000,B 0.000,C 180.000} C_DIS
LIN {X 117.455,Y 125.923,Z 52.000,A 180.000,B 0.000,C 180.000} C_DIS
LIN {X 117.098,Y 125.866,Z 52.000,A 180.000,B 0.000,C 180.000} C_DIS
LIN {X 117.056,Y 125.857,Z 52.000,A 180.000,B 0.000,C 180.000} C_DIS
LIN {X 116.740,Y 125.787,Z 52.000,A 180.000,B 0.000,C 180.000} C_DIS
LIN {X 116.561,Y 125.742,Z 52.000,A 180.000,B 0.000,C 180.000} C_DIS
LIN {X 116.204,Y 125.638,Z 52.000,A 180.000,B 0.000,C 180.000} C_DIS
LIN {X 116.025,Y 125.575,Z 52.000,A 180.000,B 0.000,C 180.000} C_DIS
LIN {X 115.816,Y 125.500,Z 52.000,A 180.000,B 0.000,C 180.000} C_DIS
LIN {X 115.667,Y 125.441,Z 52.000,A 180.000,B 0.000,C 180.000} C_DIS
LIN {X 115.310,Y 125.286,Z 52.000,A 180.000,B 0.000,C 180.000} C_DIS
LIN {X 115.131,Y 125.195,Z 52.000,A 180.000,B 0.000,C 180.000} C_DIS
LIN {X 114.952,Y 125.104,Z 52.000,A 180.000,B 0.000,C 180.000} C_DIS
LIN {X 114.774,Y 125.004,Z 52.000,A 180.000,B 0.000,C 180.000} C_DIS
LIN {X 114.595,Y 124.898,Z 52.000,A 180.000,B 0.000,C 180.000} C_DIS
LIN {X 114.416,Y 124.787,Z 52.000,A 180.000,B 0.000,C 180.000} C_DIS
LIN {X 114.150,Y 124.606,Z 52.000,A 180.000,B 0.000,C 180.000} C_DIS
LIN {X 114.058,Y 124.540,Z 52.000,A 180.000,B 0.000,C 180.000} C_DIS
LIN {X 113.880,Y 124.402,Z 52.000,A 180.000,B 0.000,C 180.000} C_DIS
LIN {X 113.701,Y 124.261,Z 52.000,A 180.000,B 0.000,C 180.000} C_DIS
LIN {X 113.484,Y 124.070,Z 52.000,A 180.000,B 0.000,C 180.000} C_DIS
LIN {X 113.343,Y 123.943,Z 52.000,A 180.000,B 0.000,C 180.000} C_DIS
LIN {X 113.112,Y 123.712,Z 52.000,A 180.000,B 0.000,C 180.000} C_DIS
LIN {X 112.986,Y 123.579,Z 52.000,A 180.000,B 0.000,C 180.000} C_DIS
LIN {X 112.788,Y 123.354,Z 52.000,A 180.000,B 0.000,C 180.000} C_DIS
LIN {X 112.641,Y 123.176,Z 52.000,A 180.000,B 0.000,C 180.000} C_DIS
LIN {X 112.450,Y 122.928,Z 52.000,A 180.000,B 0.000,C 180.000} C_DIS
LIN {X 112.373,Y 122.818,Z 52.000,A 180.000,B 0.000,C 180.000} C_DIS
LIN {X 112.251,Y 122.639,Z 52.000,A 180.000,B 0.000,C 180.000} C_DIS
LIN {X 112.135,Y 122.461,Z 52.000,A 180.000,B 0.000,C 180.000} C_DIS
LIN {X 112.029,Y 122.282,Z 52.000,A 180.000,B 0.000,C 180.000} C_DIS
LIN {X 111.924,Y 122.103,Z 52.000,A 180.000,B 0.000,C 180.000} C_DIS
LIN {X 111.734,Y 121.731,Z 52.000,A 180.000,B 0.000,C 180.000} C_DIS
LIN {X 111.660,Y 121.567,Z 52.000,A 180.000,B 0.000,C 180.000} C_DIS
LIN {X 111.556,Y 121.325,Z 52.000,A 180.000,B 0.000,C 180.000} C_DIS
LIN {X 111.509,Y 121.209,Z 52.000,A 180.000,B 0.000,C 180.000} C_DIS
LIN {X 111.377,Y 120.841,Z 52.000,A 180.000,B 0.000,C 180.000} C_DIS
LIN {X 111.326,Y 120.673,Z 52.000,A 180.000,B 0.000,C 180.000} C_DIS
LIN {X 111.274,Y 120.494,Z 52.000,A 180.000,B 0.000,C 180.000} C_DIS
LIN {X 111.226,Y 120.315,Z 52.000,A 180.000,B 0.000,C 180.000} C_DIS
LIN {X 111.146,Y 119.958,Z 52.000,A 180.000,B 0.000,C 180.000} C_DIS
LIN {X 111.114,Y 119.779,Z 52.000,A 180.000,B 0.000,C 180.000} C_DIS
LIN {X 111.086,Y 119.600,Z 52.000,A 180.000,B 0.000,C 180.000} C_DIS
LIN {X 111.059,Y 119.422,Z 52.000,A 180.000,B 0.000,C 180.000} C_DIS
LIN {X 111.019,Y 119.006,Z 52.000,A 180.000,B 0.000,C 180.000} C_DIS
LIN {X 111.013,Y 118.885,Z 52.000,A 180.000,B 0.000,C 180.000} C_DIS
LIN {X 111.002,Y 118.528,Z 52.000,A 180.000,B 0.000,C 180.000} C_DIS
LIN {X 111.006,Y 118.349,Z 52.000,A 180.000,B 0.000,C 180.000} C_DIS
LIN {X 111.012,Y 118.170,Z 52.000,A 180.000,B 0.000,C 180.000} C_DIS
LIN {X 111.019,Y 117.994,Z 52.000,A 180.000,B 0.000,C 180.000} C_DIS
LIN {X 111.053,Y 117.634,Z 52.000,A 180.000,B 0.000,C 180.000} C_DIS
LIN {X 111.077,Y 117.455,Z 52.000,A 180.000,B 0.000,C 180.000} C_DIS
LIN {X 111.134,Y 117.098,Z 52.000,A 180.000,B 0.000,C 180.000} C_DIS
LIN {X 111.173,Y 116.919,Z 52.000,A 180.000,B 0.000,C 180.000} C_DIS
LIN {X 111.213,Y 116.740,Z 52.000,A 180.000,B 0.000,C 180.000} C_DIS
LIN {X 111.258,Y 116.561,Z 52.000,A 180.000,B 0.000,C 180.000} C_DIS
LIN {X 111.362,Y 116.204,Z 52.000,A 180.000,B 0.000,C 180.000} C_DIS
LIN {X 111.377,Y 116.159,Z 52.000,A 180.000,B 0.000,C 180.000} C_DIS
LIN {X 111.489,Y 115.846,Z 52.000,A 180.000,B 0.000,C 180.000} C_DIS
LIN {X 111.556,Y 115.675,Z 52.000,A 180.000,B 0.000,C 180.000} C_DIS
LIN {X 111.714,Y 115.310,Z 52.000,A 180.000,B 0.000,C 180.000} C_DIS
LIN {X 111.734,Y 115.269,Z 52.000,A 180.000,B 0.000,C 180.000} C_DIS
LIN {X 111.913,Y 114.918,Z 52.000,A 180.000,B 0.000,C 180.000} C_DIS
LIN {X 111.996,Y 114.774,Z 52.000,A 180.000,B 0.000,C 180.000} C_DIS
LIN {X 112.102,Y 114.595,Z 52.000,A 180.000,B 0.000,C 180.000} C_DIS
LIN {X 112.213,Y 114.416,Z 52.000,A 180.000,B 0.000,C 180.000} C_DIS
LIN {X 112.335,Y 114.237,Z 52.000,A 180.000,B 0.000,C 180.000} C_DIS
LIN {X 112.450,Y 114.072,Z 52.000,A 180.000,B 0.000,C 180.000} C_DIS
LIN {X 112.628,Y 113.841,Z 52.000,A 180.000,B 0.000,C 180.000} C_DIS
LIN {X 112.739,Y 113.701,Z 52.000,A 180.000,B 0.000,C 180.000} C_DIS
LIN {X 112.986,Y 113.421,Z 52.000,A 180.000,B 0.000,C 180.000} C_DIS
LIN {X 113.057,Y 113.343,Z 52.000,A 180.000,B 0.000,C 180.000} C_DIS
LIN {X 113.343,Y 113.057,Z 52.000,A 180.000,B 0.000,C 180.000} C_DIS
LIN {X 113.421,Y 112.986,Z 52.000,A 180.000,B 0.000,C 180.000} C_DIS
LIN {X 113.701,Y 112.739,Z 52.000,A 180.000,B 0.000,C 180.000} C_DIS
LIN {X 113.841,Y 112.628,Z 52.000,A 180.000,B 0.000,C 180.000} C_DIS
LIN {X 114.072,Y 112.450,Z 52.000,A 180.000,B 0.000,C 180.000} C_DIS
LIN {X 114.237,Y 112.335,Z 52.000,A 180.000,B 0.000,C 180.000} C_DIS
LIN {X 114.416,Y 112.213,Z 52.000,A 180.000,B 0.000,C 180.000} C_DIS
LIN {X 114.494,Y 112.165,Z 52.000,A 180.000,B 0.000,C 180.000} C_DIS
; Lead Out Move Starts
LIN {X 114.952,Y 112.128,Z 52.000,A 180.000,B 0.000,C 180.000} C_DIS
LIN {X 115.247,Y 112.481,Z 52.000,A 180.000,B 0.000,C 180.000} C_DIS
LIN {X 115.444,Y 113.374,Z 52.000,A 180.000,B 0.000,C 180.000} C_DIS
LIN {X 115.521,Y 113.719,Z 52.146,A 180.000,B 0.000,C 180.000} C_DIS
LIN {X 115.552,Y 113.862,Z 52.500,A 180.000,B 0.000,C 180.000} C_DIS
; Rapid Move Starts
LIN {X 115.552,Y 113.862,Z 105.000,A 180.000,B 0.000,C 180.000} C_DIS
;ENDFOLD
END

--- sKontur5.dat ---
&ACCESS RVO
DEFDAT sKontur5
;FOLD EXTERNAL DECLARATIONS;%{PE}%MKUKATPBASIS,%CEXT,%VCOMMON,%P
  ;FOLD BASISTECH EXT;%{PE}%MKUKATPBASIS,%CEXT,%VEXT,%P
    EXT  BAS (BAS_COMMAND  :IN,REAL  :IN )
  ;ENDFOLD (BASISTECH EXT)

;ENDFOLD (EXTERNAL DECLARATIONS)
ENDDAT
